# B&R Automation Studio project Nitto (part 15)

#### FB_CrossCutter.st
```iecst
//(********************************************************************
// * COPYRIGHT -- Microsoft
// ********************************************************************
// * Programm: MAIN
// * Datei: FB_CuttingAxis.st
// * Autor: Awalz
// * Erstellt: 19. Mai 2014
// ********************************************************************
// * Implementierung des Programms MAIN
// ********************************************************************)
//
// (*<$Description$> TODO: Bitte Kommentar hier einzufügen </$Description$>*)
FUNCTION_BLOCK FB_CrossCutter
	SetupPar.Acceleration	:= 1000000.0;
	SetupPar.Deceleration	:= 1000000.0;
	SetupPar.Velocity		:= SLS_MASTER_VELO;
	RegMarkPar.WindowNegative	:= 30000.0;
	RegMarkPar.WindowPositive	:= 30000.0;

	MC_BR_ReadAxisError_0.Axis				:= SlaveREF;
	MC_BR_ReadAxisError_0.Enable			:= NOT MC_BR_ReadAxisError_0.Error;
	MC_BR_ReadAxisError_0();

	MC_ReadStatus_0.Axis					:= SlaveREF;
	MC_ReadStatus_0.Enable					:= NOT MC_ReadStatus_0.Error;
	MC_ReadStatus_0();
	MC_BR_ReadDriveStatus_0.Axis			:= SlaveREF;
	MC_BR_ReadDriveStatus_0.AdrDriveStatus	:= ADR(DriveStatus);
	MC_BR_ReadDriveStatus_0.Enable			:= NOT MC_BR_ReadDriveStatus_0.Error;
	MC_BR_ReadDriveStatus_0();

	MC_ReadActualPosition_0.Axis			:= SlaveREF;
	MC_ReadActualPosition_0.Enable			:= Enable;
	MC_ReadActualPosition_0();

	MC_Reset_0.Axis	:= SlaveREF;
	MC_Reset_0();

	MC_ReadParameter_AxisPeriod.Axis			:= SlaveREF;
	MC_ReadParameter_AxisPeriod.ParameterNumber	:= 1008;	//axis modulo period
	MC_ReadParameter_AxisPeriod.Enable			:= Enable;
	MC_ReadParameter_AxisPeriod();

//********************		CrossCutter			********************
	MC_BR_CrossCutterControl_0.Master									:= machineMaster.AxisREF;
	MC_BR_CrossCutterControl_0.Slave									:= SlaveREF;
	MC_BR_CrossCutterControl_0.CutRangeMaster 							:= crosscuttpar.CutRangeMaster;
	MC_BR_CrossCutterControl_0.CutRangeSlave 							:= crosscuttpar.CutRangeSlave;
	MC_BR_CrossCutterControl_0.ProductLength 							:= crosscuttpar.ProductLength;
	MC_BR_CrossCutterControl_0.AdvancedParameters.StartMode 			:= crosscuttpar.StartMode;
	MC_BR_CrossCutterControl_0.AdvancedParameters.StartInterval			:= crosscuttpar.StartInterval;
//    MC_BR_CrossCutterControl_0.AdvancedParameters.MasterStartDistance	:= crosscuttpar.MasterStartDistance;
//	MC_BR_CrossCutterControl_0();

	IF (MC_ReadParameter_AxisPeriod.Value <> 0.0) THEN
		NeutralPosition	:= fmod( (MC_BR_CrossCutterControl_0.AdvancedParameters.CutPosition + MC_ReadParameter_AxisPeriod.Value / 2.0), MC_ReadParameter_AxisPeriod.Value);
//		IS.NeutralPosition	:= 0.0;			// Stanze ist nach Referenzfahrt in Position
	ELSE
		NeutralPosition	:= 0.0;
	END_IF;

	//**********************	START OF STATE MACHINE	**************************
	//**********************	transitions from any state	**********************
	IF (NOT Enable) THEN
		Error		:= FALSE;
		ErrorID		:= 0;
		State	:= STATE_DISABLED;
//	ELSIF (markpoints.Error) THEN
//		ErrorID		:= markpoints.ErrorID;
//		Error		:= TRUE;
//		State	:= STATE_ERROR;
	ELSIF (MC_BR_CrossCutterControl_0.Error) THEN
		ErrorID		:= MC_BR_CrossCutterControl_0.ErrorID;
		Error		:= TRUE;
		State	:= STATE_ERROR;
//	ELSIF (MC_BR_Phasing_0.Error) THEN
//		ErrorID		:= MC_BR_Phasing_0.ErrorID;
//		Error		:= TRUE;
//		State	:= STATE_ERROR;
//	ELSIF (MC_BR_ReadAutPosition_0.Error) THEN
//		ErrorID		:= MC_BR_ReadAutPosition_0.ErrorID;
//		Error		:= TRUE;
//		State	:= STATE_ERROR;
	ELSIF (MC_MoveAbsolute_0.Error) THEN
		ErrorID		:= MC_MoveAbsolute_0.ErrorID;
		Error		:= TRUE;
		State	:= STATE_ERROR;
	ELSIF (MC_ReadParameter_AxisPeriod.Error) THEN
		ErrorID		:= MC_ReadParameter_AxisPeriod.ErrorID;
		Error		:= TRUE;
		State	:= STATE_ERROR;
	END_IF;
	//****************************************************************************

	CASE State OF
		//**********************	FUB inactive	**********************
		STATE_DISABLED:
			MC_BR_ReadAutPosition_0.Execute		:= FALSE;
			MC_MoveAbsolute_0.Execute			:= FALSE;
			MC_BR_CrossCutterControl_0.Enable	:= FALSE;
			MC_BR_CrossCutterControl_0.EnableCut:= FALSE;
			EnableRestart						:= FALSE;
			SetupComplete						:= FALSE;

			IF Enable  (*OR RestartAllowed *)THEN
				State	:= STATE_INIT;
			END_IF;
	//****************************************************************

	//**********************	Internal variables are initialized	**********************
		STATE_INIT:
			GetNextCuttPos.reset := TRUE;
			State	:= STATE_IDLE;
	//************************************************************************************

	//**********************	Waiting for a movement command	**********************
		STATE_IDLE:
			GetNextCuttPos.reset := FALSE;
			IF RestartAllowed THEN
				EnableRestart						:= TRUE;
			END_IF;
			IF (EnableMove) THEN
				MC_BR_CrossCutterControl_0.Enable	:= TRUE;
				MC_BR_CrossCutterControl_0.EnableCut:= FALSE;
				State	:= STATE_CHECK_STANDBY;
			END_IF;
	//*********************************************************************************

	//**********************	Checking if automat restart is possible	**********************
		STATE_CHECK_STANDBY:
			IF (MC_BR_CrossCutterControl_0.Active) THEN
				MC_BR_CrossCutterControl_0.Enable		:= FALSE;
				MC_BR_CrossCutterControl_0.EnableCut	:= FALSE;
				IF (MC_BR_CrossCutterControl_0.StandBy AND EnableRestart) THEN
					MC_BR_ReadAutPosition_0.Execute		:= TRUE;
					State	:= STATE_READ_AUT_POS;
				ELSE
					SetupComplete					:= FALSE;
					MC_MoveAbsolute_0.Direction		:= mcPOSITIVE_DIR;
					MC_MoveAbsolute_0.Position		:= NeutralPosition;
					//IS.MC_MoveAbsolute_0.Execute		:= TRUE;	// Keine Bewegung mehr auf die NeutralPosition
					// 2013-08-22 /scoenefeldr/
				(*	MC_BR_CrossCutterControl_0.AdvancedParameters.MasterStartDistance	:= MC_BR_CrossCutterControl_0.AdvancedParameters.CutPosition - MC_ReadActualPosition_0.Position;*)
						MC_BR_CrossCutterControl_0.AdvancedParameters.MasterStartDistance	:= MC_BR_CrossCutterControl_0.AdvancedParameters.CutPosition + MC_ReadActualPosition_0.Position;
					IF (MC_BR_CrossCutterControl_0.AdvancedParameters.MasterStartDistance < 0 OR MC_BR_CrossCutterControl_0.AdvancedParameters.MasterStartDistance < data.general.periodLength) THEN
						MC_BR_CrossCutterControl_0.AdvancedParameters.MasterStartDistance	:= (*MC_BR_CrossCutterControl_0.AdvancedParameters.MasterStartDistance + *)data.general.periodLength;
					ELSIF (MC_BR_CrossCutterControl_0.AdvancedParameters.MasterStartDistance > data.general.periodLength) THEN
						MC_BR_CrossCutterControl_0.AdvancedParameters.MasterStartDistance	:=(* MC_BR_CrossCutterControl_0.AdvancedParameters.MasterStartDistance - data.general.periodLength;*) scalePerimeter.realperimeter;
					END_IF
					State							:= STATE_MOVE_TO_NEUTRAL_POS;
				END_IF;
			END_IF;
			IF (NOT EnableMove) THEN
				MC_BR_ReadAutPosition_0.Execute		:= FALSE;
				MC_BR_CrossCutterControl_0.Enable	:= FALSE;
				MC_BR_CrossCutterControl_0.EnableCut:= FALSE;
				State	:= STATE_IDLE;
			END_IF;
	//****************************************************************************************

	//**********************	Reading automat position	**********************
		STATE_READ_AUT_POS:
			IF (MC_BR_ReadAutPosition_0.Done) THEN
				MC_BR_ReadAutPosition_0.Execute	:= FALSE;
				MC_MoveAbsolute_0.Direction		:= mcPOSITIVE_DIR + mcAUTOMAT_POS;
				MC_MoveAbsolute_0.Position		:= MC_BR_ReadAutPosition_0.AutPosition;
				MC_MoveAbsolute_0.Execute		:= TRUE;
				State							:= STATE_MOVE_TO_AUT_POS;
			END_IF;

			IF (NOT EnableMove) THEN
				MC_BR_ReadAutPosition_0.Execute	:= FALSE;
				MC_MoveAbsolute_0.Execute		:= FALSE;
				State	:= STATE_IDLE;
			END_IF;
	//*****************************************************************************

	//**********************	Moving to automat position	**********************
		STATE_MOVE_TO_AUT_POS:
			IF MC_MoveAbsolute_0.Done THEN
				MC_MoveAbsolute_0.Execute			:= FALSE;
				MC_BR_CrossCutterControl_0.AdvancedParameters.StartMode	:= mcRESTART + mcCORRECT_CURRENT_CYCLE;
				MC_BR_CrossCutterControl_0.Enable	:= TRUE;
				MC_BR_CrossCutterControl_0.EnableCut:= TRUE;
				MC_BR_CrossCutterControl_0.AdvancedParameters.MasterMaxVelocity	:= SetupPar.Velocity; (*data.general.maxVelocity;*)
				State	:= STATE_START_AUTOMAT;
			ELSIF MC_MoveAbsolute_0.CommandAborted THEN
				MC_MoveAbsolute_0.Execute			:= FALSE;
				State	:= STATE_W4_RESET;
			END_IF;

			IF NOT EnableMove THEN
				MC_MoveAbsolute_0.Execute			:= FALSE;
				MC_BR_CrossCutterControl_0.Enable	:= FALSE;
				MC_BR_CrossCutterControl_0.EnableCut:= FALSE;
				State	:= STATE_IDLE;
			END_IF;
	//*****************************************************************************

	//**********************	Moving to neutral position	**********************
		STATE_MOVE_TO_NEUTRAL_POS:
			IF (TRUE) THEN
				MC_MoveAbsolute_0.Execute			:= FALSE;
				MC_BR_CrossCutterControl_0.AdvancedParameters.StartMode	:= mcIMMEDIATE + mcCORRECT_CURRENT_CYCLE;
				MC_BR_CrossCutterControl_0.Enable	:= TRUE;
				MC_BR_CrossCutterControl_0.EnableCut:= TRUE;
				MC_BR_CrossCutterControl_0.AdvancedParameters.MasterMaxVelocity	:= SetupPar.Velocity; (*data.general.maxVelocity;*)
				State	:= STATE_START_AUTOMAT;

			ELSIF (MC_MoveAbsolute_0.CommandAborted) THEN
				MC_MoveAbsolute_0.Execute	:= FALSE;
				State	:= STATE_W4_RESET;
			END_IF;

			IF NOT EnableMove THEN
				MC_MoveAbsolute_0.Execute			:= FALSE;
				MC_BR_CrossCutterControl_0.Enable	:= FALSE;
				MC_BR_CrossCutterControl_0.EnableCut:= FALSE;
				State	:= STATE_IDLE;
			END_IF;
	//*****************************************************************************

	//**********************	Starting cam automat	**********************
		STATE_START_AUTOMAT:
			IF (MC_BR_CrossCutterControl_0.Active) THEN
				EnableRestart	:= TRUE;
				State			:= STATE_RUNNING;
			ELSIF (MC_BR_CrossCutterControl_0.CommandAborted) THEN
				MC_BR_CrossCutterControl_0.Enable	:= FALSE;
				MC_BR_CrossCutterControl_0.EnableCut:= FALSE;
				State	:= STATE_W4_RESET;
			END_IF;

			IF (NOT EnableMove) THEN
				MC_BR_CrossCutterControl_0.Enable	:= FALSE;
				MC_BR_CrossCutterControl_0.EnableCut:= FALSE;
				State	:= STATE_IDLE;
			END_IF;
	//************************************************************************

	//**********************	Cam automat is running	**********************
		STATE_RUNNING:
			IF (MC_BR_CrossCutterControl_0.CommandAborted) THEN
				MC_BR_CrossCutterControl_0.Enable	:= FALSE;
				MC_BR_CrossCutterControl_0.EnableCut:= FALSE;
				State	:= STATE_W4_RESET;
			END_IF;
//			IF RestartAllowed THEN (* um die Achse wieder zu koppeln*)
//				RestartAllowed := FALSE;
//				EnableRestart						:= TRUE;
//				MC_BR_CrossCutterControl_0.Enable	:= FALSE;
//				MC_BR_CrossCutterControl_0.EnableCut:= FALSE;
//				State	:= STATE_W4_RESET;
//			END_IF
			//cam automat synchronization movement is complete
			IF ( (MC_BR_CrossCutterControl_0.IS.AutActStIdx >= 2) AND (MC_BR_CrossCutterControl_0.IS.AutActStIdx <= 6) ) THEN
				SetupComplete	:= TRUE;
			END_IF;
			//set master speed to maximum velocity after start movement is complete
			IF (MC_BR_CrossCutterControl_0.InCompensation) THEN
				MC_BR_CrossCutterControl_0.AdvancedParameters.MasterMaxVelocity	:= SetupPar.Velocity; (*data.general.maxVelocity;;*)
			END_IF;
			IF (NOT EnableMove) THEN
				MC_BR_CrossCutterControl_0.Enable	:= FALSE;
				MC_BR_CrossCutterControl_0.EnableCut	:= FALSE;
			State	:= STATE_IDLE;
			END_IF;
	//************************************************************************

	//**********************	Command aborted, wait until "EnableMove" is reset	**********************
		STATE_W4_RESET:
			IF  EnableMove THEN
				State	:= STATE_IDLE;
			END_IF;
	//************************************************************************

	//**********************	FUB Error	**********************
		STATE_ERROR:
			(*MC_BR_CrossCutterControl_0.AdvancedParameters.MasterStartDistance	:= 0;*)
			MC_BR_CrossCutterControl_0.Enable := FALSE;
			State := STATE_CHECK_STANDBY;
	//************************************************************

		ELSE

	END_CASE;
	//**********************	END OF STATE MACHINE	************************

	(*********************		Read automat position	********************)
	MC_BR_ReadAutPosition_0.Axis		:= SlaveREF;
	MC_BR_ReadAutPosition_0();
	//******************************************************************************
	//********************		Move absolute			********************
	MC_MoveAbsolute_0.Axis			:= SlaveREF;
	MC_MoveAbsolute_0.Velocity		:= 40000;
	MC_MoveAbsolute_0.Acceleration	:= 60000;
	MC_MoveAbsolute_0.Deceleration	:= 60000;
	MC_MoveAbsolute_0();
	//*********************************************************************

	//**************************************************************************//
	//limit correction value
	LCRLimit_Correction.max_value	:= REAL_TO_DINT (data.recipe.MaxCorr);  (*AutPar.MaxCorrection;*)
	LCRLimit_Correction.min_value	:= - REAL_TO_DINT (data.recipe.MaxCorr); (* AutPar.MaxCorrection;*)

	//calculate cut position within tool segment period
	IF (MC_ReadParameter_AxisPeriod.Value <> 0.0) THEN
		MC_BR_CrossCutterControl_0.CutRangeSlave		:= DINT_TO_REAL( (crosscuttpar.CutEndPos - crosscuttpar.CutStartPos) MOD REAL_TO_DINT(MC_ReadParameter_AxisPeriod.Value) );
		IF (MC_BR_CrossCutterControl_0.CutRangeSlave < 0.0) THEN
			MC_BR_CrossCutterControl_0.CutRangeSlave	:= MC_BR_CrossCutterControl_0.CutRangeSlave + MC_ReadParameter_AxisPeriod.Value;
		END_IF
		IF 	crosscuttpar.CutStartPos > crosscuttpar.CutEndPos THEN
			MC_BR_CrossCutterControl_0.AdvancedParameters.CutPosition	:= DINT_TO_REAL((crosscuttpar.CutEndPos + crosscuttpar.CutStartPos + REAL_TO_DINT(MC_ReadParameter_AxisPeriod.Value)) / 2 MOD REAL_TO_DINT(MC_ReadParameter_AxisPeriod.Value));
		ELSE
			MC_BR_CrossCutterControl_0.AdvancedParameters.CutPosition	:= DINT_TO_REAL((crosscuttpar.CutEndPos + crosscuttpar.CutStartPos) /2 MOD REAL_TO_DINT(MC_ReadParameter_AxisPeriod.Value));
		END_IF
			IF (MC_BR_CrossCutterControl_0.AdvancedParameters.CutPosition < 0.0) THEN
			MC_BR_CrossCutterControl_0.AdvancedParameters.CutPosition	:= MC_BR_CrossCutterControl_0.AdvancedParameters.CutPosition + MC_ReadParameter_AxisPeriod.Value;
			END_IF;
		//limit cut range of slave to avoid ACOPOS errors on wrong user input
		IF ((crosscuttpar.MinCutRangeSlave > 0.0) AND (crosscuttpar.MinCutRangeSlave < MC_ReadParameter_AxisPeriod.Value)) THEN
			MC_BR_CrossCutterControl_0.CutRangeSlave	:= MAX(MC_BR_CrossCutterControl_0.CutRangeSlave, crosscuttpar.MinCutRangeSlave);
		END_IF;
		IF ((crosscuttpar.MinCompRangeSlave > 0.0) AND (crosscuttpar.MinCompRangeSlave < MC_ReadParameter_AxisPeriod.Value) ) THEN
			MC_BR_CrossCutterControl_0.CutRangeSlave := MIN(MC_BR_CrossCutterControl_0.CutRangeSlave, (MC_ReadParameter_AxisPeriod.Value - crosscuttpar.MinCompRangeSlave));
		END_IF;

		//scale cut range of master
		LCRLimScal_CutRangeMaster.x1	:= 0.0;
		LCRLimScal_CutRangeMaster.y1	:= MC_BR_CrossCutterControl_0.CutRangeSlave;
		LCRLimScal_CutRangeMaster.x2	:= 100.0;
		LCRLimScal_CutRangeMaster.y2	:= (MC_BR_CrossCutterControl_0.CutRangeSlave * crosscuttpar.ProductLength) / MC_ReadParameter_AxisPeriod.Value;
		LCRLimScal_CutRangeMaster.x		:= crosscuttpar.Insetting;
		LCRLimScal_CutRangeMaster();
		MC_BR_CrossCutterControl_0.CutRangeMaster	:= LCRLimScal_CutRangeMaster.y;
	ELSE
		MC_BR_CrossCutterControl_0.CutRangeSlave					:= 0.0;
		MC_BR_CrossCutterControl_0.CutRangeMaster					:= 0.0;
		MC_BR_CrossCutterControl_0.AdvancedParameters.CutPosition	:= 0.0;
	END_IF;
	//******************************************************************
	//choose source of reg mark correction
	GetNextCuttPos( scalePerimeter := scalePerimeter, markpoints := markpoints, machinemaster := machineMaster);

	IF (RegMarkPar.EnableRmCorrection) THEN
		IF (RegMarkPar.EnableVRegMark) THEN
			LCRLimit_Correction.in	:= GetNextCuttPos.setCutOffset.setOffset_o;
			syncFtrig(CLK := MC_BR_CrossCutterControl_0.InCut);
			IF syncFtrig.Q THEN
				initdata := TRUE;
			END_IF
			(*Steckung bzw. Stauchung der Länge;*)
			IF MC_BR_CrossCutterControl_0.CutCount  <>  CutCount_1 AND initdata THEN
				CutCount_1 := MC_BR_CrossCutterControl_0.CutCount;
				MC_BR_CrossCutterControl_0.InitData	:= TRUE;
				initdata := FALSE;
			END_IF
		ELSE
			LCRLimit_Correction.in	:= GetNextCuttPos.PositionError;
//			syncFtrig(CLK := MC_BR_CrossCutterControl_0.InCut);
//			IF syncFtrig.Q THEN
//				initdata := TRUE;
//			END_IF

			syncRtrig(CLK := MC_BR_CrossCutterControl_0.InCut);
			IF MC_BR_CrossCutterControl_0.CutCount <> CutCntOld THEN
				initdata := TRUE;
				CutCntOld := MC_BR_CrossCutterControl_0.CutCount;
			END_IF
			IF  markpoints.ProbeCounter  <>  CutCount_1 AND markpoints.ProbeCounter < 1 AND initdata THEN
				CutCount_1 := markpoints.ProbeCounter;
				MC_BR_CrossCutterControl_0.InitData	:= TRUE;
				initdata := FALSE;
			ELSIF markpoints.ProbeCounter > 1 AND initdata THEN
				MC_BR_CrossCutterControl_0.InitData	:= TRUE;
				initdata := FALSE;
			END_IF
//			R_TRIG_InCompensation(CLK := MC_BR_CrossCutterControl_0.InCompensation);
//			IF R_TRIG_InCompensation.Q THEN
//				initdata := TRUE;
//			END_IF
//			IF  GetNextCuttPos.newdata <>  CutCount_1 AND  NOT MC_BR_CrossCutterControl_0.InCut(*AND initdata*) THEN
//				CutCount_1 := GetNextCuttPos.newdata;
//				MC_BR_CrossCutterControl_0.InitData	:= TRUE;
//				initdata := FALSE;
//			END_IF
		END_IF;
	ELSE
		LCRLimit_Correction.in	:= 0.0;
	END_IF;
	LCRLimit_Correction();	(*markpoints.CorrectionValid *)
	MC_BR_CrossCutterControl_0.ProductLengthCorrection	:= LCRLimit_Correction.out;
	IF MC_BR_CrossCutterControl_0.InitData THEN
		(*MC_BR_CrossCutterControl_0.ProductLengthCorrection	:= LCRLimit_Correction.out;*)
		OffsetValue1 := REAL_TO_DINT (MC_BR_CrossCutterControl_0.ProductLengthCorrection);
	END_IF
	MC_BR_CrossCutterControl_0();
	markpoints();
	IF MC_BR_CrossCutterControl_0.DataInitialized THEN
		MC_BR_CrossCutterControl_0.InitData	:= FALSE;
	END_IF
	Active				:= MC_BR_CrossCutterControl_0.Active;
	CutMasterPosition	:= MC_BR_CrossCutterControl_0.CutMasterPosition;
	RegMarkPar.Axis 	:= SlaveREF;
	//probe counter
	(*markpoints();*)
	ProbeCounter		:= markpoints.ProbeCounter;
	MissedTriggers		:= markpoints.MissedTriggers;
	ActPositionError	:= markpoints.CorrectionValue;
	IF (Enable AND RegMarkPar.EnableRmCorrection) THEN
		IF (RegMarkPar.EnableVRegMark) THEN
			ProbeCounter		:= ProbeCounter + BOOL_TO_UDINT(SPR_RmCalcPosError_Virtual.RecordedValueValid);
			MissedTriggers		:= 0;
			ActPositionError	:= PositionError;
		ELSE

		END_IF;
	ELSE
		ProbeCounter		:= 0;
		MissedTriggers		:= 0;
		ActPositionError	:= 0;
	END_IF;
END_FUNCTION_BLOCK
```

#### ac_manualCU.st
```iecst
(********************************************************************
 * COPYRIGHT -- Microsoft
 ********************************************************************
 * Programm: MAIN
 * Datei: ac_manualCU.st
 * Autor: Awalz
 * Erstellt: 21. Mai 2014
 ********************************************************************
 * Implementierung des Programms MAIN
 ********************************************************************)

 (*<$Description$> Fügt eine neue Aktion zum IEC Programm oder Bibliothek </$Description$>*)
ACTION ac_manualCU:
	status.isCoupled := axis.ctrl.MC_ReadStatus_0.SynchronizedMotion;

	CASE state OF
		ST_IDLE:

			IF status.dataOk THEN
				IF data.newTools OR data.newRecipe THEN
					IF data.recipe.mode = CONST.CUTTINGUNIT.MODEs.DISABLE THEN
						modeCtrl.mode := data.recipe.mode;
						config (cmd := CONST.CUTTINGUNIT.CMDs.DEINIT, machineMaster := machineMaster,axis := axis, status := status, data := data,
						IOs := IOs, powerbridge := powerbridge, scalePerimeter := scalePerimeter,markpoints := markpoints, camtable := camtable,  getNextUnitSyncPos := getNextUnitSyncPos, setCutOffset := setCutOffset);
						busy := TRUE;
						state := ST_SETDATA_WAIT;
					ELSE
						modeCtrl.mode := data.recipe.mode;
						check(machdata := data.machdata, recipe := data.recipe, general := data.general, modeCtrl := modeCtrl);
						IF check.err.flag THEN
							data.err := check.err;
						ELSE
							config (cmd := CONST.CUTTINGUNIT.CMDs.SETDATA, machineMaster := machineMaster, axis := axis, status := status, data := data,
							IOs := IOs, powerbridge := powerbridge, scalePerimeter := scalePerimeter,markpoints := markpoints, camtable := camtable,  getNextUnitSyncPos := getNextUnitSyncPos, setCutOffset := setCutOffset);
							state := ST_SETDATA_WAIT;
						END_IF
					END_IF
				ELSE
					IF data.recipe.mode = CONST.CUTTINGUNIT.MODEs.DISABLE THEN // Stanzen dennoch bewegen können*)

						IF cmdCtrl.value = CONST.CUTTINGUNIT.CMDs.MOVEFW OR cmdCtrl.value = CONST.CUTTINGUNIT.CMDs.MOVEBW THEN
							cmdStatus(set := TRUE, value := cmdCtrl.value);
							busy := TRUE;
							state := ST_MOVE_START;
						ELSIF cmdCtrl.value <> CONST.CUTTINGUNIT.CMDs.NO_CMD AND NOT cmdCtrl.value = CONST.CUTTINGUNIT.CMDs.RESET THEN
							cmdStatus(set := TRUE, value := cmdCtrl.value);
							busy := TRUE;
							state := ST_FUNCTION_START;
						END_IF
					ELSE
						IF NOT status.isCalibrated OR NOT axis.ctrl.BasicControl.AxisState.Homed THEN
							modeCtrl.mode := data.recipe.mode;
							IF cmdCtrl.value = CONST.CUTTINGUNIT.CMDs.CALIBR THEN (*warten bis das kommando  gesetzt wird*)
								cmdStatus(set := TRUE, value := cmdCtrl.value);
								busy := TRUE;
								state := ST_FUNCTION_START;
							ELSIF cmdCtrl.value = CONST.CUTTINGUNIT.CMDs.MOVEFW OR cmdCtrl.value = CONST.CUTTINGUNIT.CMDs.MOVEBW THEN
								cmdStatus(set := TRUE, value := cmdCtrl.value);
								busy := TRUE;
								state := ST_MOVE_START;
							END_IF
						ELSE
							IF cmdCtrl.value = CONST.CUTTINGUNIT.CMDs.MOVEFW OR cmdCtrl.value = CONST.CUTTINGUNIT.CMDs.MOVEBW THEN
								cmdStatus(set := TRUE, value := cmdCtrl.value);
								busy := TRUE;
								state := ST_MOVE_START;
							ELSIF cmdCtrl.value = CONST.CUTTINGUNIT.CMDs.CALIBR THEN
								cmdStatus(set := TRUE, value := cmdCtrl.value);
								busy := TRUE;
								state := ST_FUNCTION_QUIT;
							ELSIF cmdCtrl.value = CONST.CUTTINGUNIT.CMDs.SYNC THEN
								cmdStatus(set := TRUE, value := cmdCtrl.value);
								busy := TRUE;
								state := ST_FUNCTION_START;
							ELSIF cmdCtrl.value = CONST.CUTTINGUNIT.CMDs.CPL_ON THEN// manuell koppeln
								cmdStatus(set := TRUE, value := cmdCtrl.value);
								busy := TRUE;
								state := ST_FUNCTION_START;
							ELSIF manualFirst AND axis.ctrl.MC_ReadStatus_0.StandStill THEN//bei Steuerung Aus/Ein wieder einkoppeln
								busy := TRUE;
								manualFirst := FALSE;
								state := ST_CPLON_WAIT;
							END_IF
						END_IF
					END_IF
				END_IF
			END_IF

		ST_CPLON_WAIT:
			IF config.busy THEN
				config(cmd := CONST.CUTTINGUNIT.CMDs.NO_CMD, machineMaster := machineMaster, axis := axis, status := status,data := data,
				IOs := IOs, powerbridge := powerbridge, scalePerimeter := scalePerimeter,markpoints := markpoints, camtable := camtable,  getNextUnitSyncPos := getNextUnitSyncPos, setCutOffset := setCutOffset);
			ELSE
				config(cmd := CONST.CUTTINGUNIT.CMDs.CPL_ON, machineMaster := machineMaster, axis := axis, status := status,data := data,
				IOs := IOs, powerbridge := powerbridge, scalePerimeter := scalePerimeter,markpoints := markpoints, camtable := camtable,  getNextUnitSyncPos := getNextUnitSyncPos, setCutOffset := setCutOffset);
				state := ST_FUNCTION;
			END_IF

		ST_SETDATA_WAIT:
			config ( machineMaster := machineMaster, axis := axis, status := status, data := data, IOs := IOs, powerbridge := powerbridge,
				scalePerimeter := scalePerimeter, markpoints := markpoints, camtable := camtable,  getNextUnitSyncPos := getNextUnitSyncPos, setCutOffset := setCutOffset);
			IF NOT config.busy THEN
				IF config.err.flag THEN
					err := config.err;
					err.state := state;
					state := ST_ERROR;
				ELSE
					tmpData(set := TRUE, setMasterModulData := data.general, setMach := data.machdata, setRecipe := data.recipe, BetrCtrl := BetrCtrl );
					data(newRecipe := FALSE, newMach := FALSE);
					busy := FALSE;
					config(cmd := CONST.CUTTINGUNIT.CMDs.NO_CMD, machineMaster := machineMaster, axis := axis, status := status,data := data,
					IOs := IOs, powerbridge := powerbridge, scalePerimeter := scalePerimeter,markpoints := markpoints, camtable := camtable,  getNextUnitSyncPos := getNextUnitSyncPos, setCutOffset := setCutOffset);
					state := ST_IDLE;
				END_IF
			ELSIF  cmdCtrl.value = CONST.CUTTINGUNIT.CMDs.RESET THEN //14.04.15
				config(cmd := CONST.CUTTINGUNIT.CMDs.RESET, machineMaster := machineMaster, axis := axis, status := status, data := data,
				IOs := IOs, powerbridge := powerbridge, scalePerimeter := scalePerimeter,markpoints := markpoints, camtable := camtable,  getNextUnitSyncPos := getNextUnitSyncPos, setCutOffset := setCutOffset);
				state := ST_FUNCTION_ABORT_WAIT;
			END_IF

		ST_FUNCTION_START:
			IF config.busy OR config.cmd <> CONST.CUTTINGUNIT.CMDs.NO_CMD THEN
				config(cmd := CONST.CUTTINGUNIT.CMDs.NO_CMD, machineMaster := machineMaster, axis := axis, status := status, data := data,
				IOs := IOs, powerbridge := powerbridge, scalePerimeter := scalePerimeter, markpoints := markpoints, camtable := camtable,  getNextUnitSyncPos := getNextUnitSyncPos, setCutOffset := setCutOffset);
			ELSE
				config (cmd := cmdStatus.value, machineMaster := machineMaster, axis := axis, status := status, data := data, IOs := IOs,
				powerbridge := powerbridge, scalePerimeter := scalePerimeter, markpoints := markpoints, camtable := camtable,  getNextUnitSyncPos := getNextUnitSyncPos, setCutOffset := setCutOffset);
				state := ST_FUNCTION;
			END_IF

		ST_FUNCTION://12
			config(machineMaster := machineMaster, axis := axis, status := status, data := data, IOs := IOs, powerbridge := powerbridge,
				scalePerimeter := scalePerimeter, markpoints := markpoints, camtable := camtable, getNextUnitSyncPos := getNextUnitSyncPos, setCutOffset := setCutOffset);
			IF cmdCtrl.value = CONST.CUTTINGUNIT.CMDs.ABORT THEN
				config(cmd := CONST.CUTTINGUNIT.CMDs.ABORT, machineMaster := machineMaster, axis := axis, status := status, data := data,
				IOs := IOs, powerbridge := powerbridge, scalePerimeter := scalePerimeter, markpoints := markpoints, camtable := camtable,  getNextUnitSyncPos := getNextUnitSyncPos, setCutOffset := setCutOffset);
				state := ST_FUNCTION_ABORT_WAIT;
			ELSIF NOT config.busy THEN
				IF config.err.flag THEN
					err := config.err;
					err.state := state;
				END_IF
				config(cmd := CONST.CUTTINGUNIT.CMDs.NO_CMD, machineMaster := machineMaster, axis := axis, status := status, data := data,
				IOs := IOs, powerbridge := powerbridge, scalePerimeter := scalePerimeter,markpoints := markpoints, camtable := camtable,  getNextUnitSyncPos := getNextUnitSyncPos, setCutOffset := setCutOffset);
				state := ST_FUNCTION_QUIT;
			ELSIF (*config.err.flag AND*) cmdCtrl.value = CONST.CUTTINGUNIT.CMDs.RESET THEN //14.04.15
				config(cmd := CONST.CUTTINGUNIT.CMDs.RESET, machineMaster := machineMaster, axis := axis, status := status, data := data,
				IOs := IOs, powerbridge := powerbridge, scalePerimeter := scalePerimeter,markpoints := markpoints, camtable := camtable,  getNextUnitSyncPos := getNextUnitSyncPos, setCutOffset := setCutOffset);
				state := ST_FUNCTION_ABORT_WAIT;
			END_IF

		ST_FUNCTION_ABORT_WAIT:
			config( machineMaster := machineMaster, axis := axis, status := status, data := data,IOs := IOs, powerbridge := powerbridge,
				scalePerimeter := scalePerimeter, markpoints := markpoints, camtable := camtable,  getNextUnitSyncPos := getNextUnitSyncPos, setCutOffset := setCutOffset);
			IF NOT config.busy THEN
				IF config.err.flag THEN
					err := config.err;
					err.state := state;
				END_IF
				config(cmd := CONST.CUTTINGUNIT.CMDs.NO_CMD, machineMaster := machineMaster, axis := axis, status := status, data := data,
				IOs := IOs, powerbridge := powerbridge, scalePerimeter := scalePerimeter,markpoints := markpoints, camtable := camtable,  getNextUnitSyncPos := getNextUnitSyncPos, setCutOffset := setCutOffset);
				state := ST_FUNCTION_QUIT;
			END_IF

		ST_FUNCTION_QUIT:
			busy := FALSE;
			IF cmdCtrl.value = CONST.CUTTINGUNIT.CMDs.NO_CMD THEN
				cmdStatus(set := TRUE, value := CONST.CUTTINGUNIT.CMDs.NO_CMD);
				state := ST_IDLE;
			END_IF

		ST_MOVE_START:

			IF config.busy OR config.cmd <> CONST.CUTTINGUNIT.CMDs.NO_CMD THEN //27.04.15
				config(cmd := CONST.CUTTINGUNIT.CMDs.NO_CMD, machineMaster := machineMaster, axis := axis, status := status, data := data, IOs := IOs, powerbridge := powerbridge,
				scalePerimeter := scalePerimeter, markpoints := markpoints, camtable := camtable, getNextUnitSyncPos := getNextUnitSyncPos,setCutOffset := setCutOffset);
			ELSIF NOT config.busy THEN //27.04.15
				config(cmd := cmdStatus.value, machineMaster := machineMaster, axis := axis, status := status, data := data, IOs := IOs, powerbridge := powerbridge,
				scalePerimeter := scalePerimeter, markpoints := markpoints, camtable := camtable,getNextUnitSyncPos := getNextUnitSyncPos,setCutOffset := setCutOffset);
				state := ST_MOVE;
			END_IF

		ST_MOVE:
			config(machineMaster := machineMaster, axis := axis, status := status, data := data, IOs := IOs, powerbridge := powerbridge,
				scalePerimeter := scalePerimeter, markpoints := markpoints, camtable := camtable,  getNextUnitSyncPos := getNextUnitSyncPos, setCutOffset := setCutOffset);
			IF cmdCtrl.value = CONST.CUTTINGUNIT.CMDs.NO_CMD THEN
				config(cmd := CONST.CUTTINGUNIT.CMDs.NO_CMD, machineMaster := machineMaster, axis := axis, status := status, data := data,
				IOs := IOs, powerbridge := powerbridge, scalePerimeter := scalePerimeter, markpoints := markpoints, camtable := camtable,  getNextUnitSyncPos := getNextUnitSyncPos, setCutOffset := setCutOffset);
				state := ST_MOVE_QUIT;

			ELSE
				config(cmd := cmdStatus.value, machineMaster := machineMaster, axis := axis, status := status, data := data,
				IOs := IOs, powerbridge := powerbridge, scalePerimeter := scalePerimeter, markpoints := markpoints,camtable := camtable,  getNextUnitSyncPos := getNextUnitSyncPos, setCutOffset := setCutOffset);
			END_IF

		ST_MOVE_QUIT:
			config(cmd := CONST.CUTTINGUNIT.CMDs.NO_CMD, machineMaster := machineMaster, axis := axis, status := status, data := data,
			IOs := IOs, powerbridge := powerbridge, scalePerimeter := scalePerimeter, markpoints := markpoints, camtable := camtable,  getNextUnitSyncPos := getNextUnitSyncPos, setCutOffset := setCutOffset);
			IF NOT config.busy THEN
				busy := FALSE;
				cmdStatus(set := TRUE, value := CONST.CUTTINGUNIT.CMDs.NO_CMD);
				state := ST_IDLE;
			ELSIF cmdCtrl.value = CONST.CUTTINGUNIT.CMDs.RESET THEN //14.04.15
				config(cmd := CONST.CUTTINGUNIT.CMDs.RESET, machineMaster := machineMaster, axis := axis, status := status, data := data,
				IOs := IOs, powerbridge := powerbridge, scalePerimeter := scalePerimeter,markpoints := markpoints, camtable := camtable,  getNextUnitSyncPos := getNextUnitSyncPos, setCutOffset := setCutOffset);
				state := ST_FUNCTION_ABORT_WAIT;
			END_IF

		ST_ERROR:
			err.set := TRUE;
			busy := FALSE;
			IF cmdCtrl.value <> CONST.CUTTINGUNIT.CMDs.NO_CMD THEN
				err(reset := TRUE);
				state := ST_IDLE;
			ELSIF BetrCtrl.value <> CONST.MACHINEMODES.MANUAL THEN
				state := ST_IDLE;
				err(reset := TRUE);
				busy := TRUE;
				StateCtrl := CTRL_MANUAL_AFTER;
			END_IF
	END_CASE

END_ACTION
```

#### ac_cyclicCuttingCtrl.st
```iecst
(********************************************************************
 * COPYRIGHT -- Microsoft
 ********************************************************************
 * Programm: MAIN
 * Datei: ac_cyclicCuttingCtrl.st
 * Autor: awalz
 * Erstellt: 25. Juli 2014
 ********************************************************************
 * Implementierung des Programms MAIN
 ********************************************************************)

(* Fügt eine neue Aktion zum IEC Programm oder Bibliothek *)
ACTION ac_cyclicCuttingCtrl:
	markpoints.TriggerInput.Edge			:= ncP_EDGE;
	markpoints.TriggerInput.EventSourceParID:= ACP10PAR_STAT_TRIGGER1;
	markpoints.TriggerInput.MaxWidth		:= 0;
	markpoints.TriggerInput.MinWidth		:= 0;
	markpoints.TriggerInput.ProbeParID		:= ACP10PAR_MA1_CYCLIC_POS;
	markpoints.TriggerInput.SensorDelay	:= -900;
//	getNextCuttPos.setCutOffset.maxcorrection :=  REAL_TO_UDINT(data.general.periodLength /2);
//	getNextCuttPos.ProductLength := REAL_TO_UDINT(data.general.periodLength);
//	getNextCuttPos.DistanceToSensor := data.machdata.position; (*540000;*)
//	axis.ctrl();
//	cmdCtrl();
//	emcy_inputs();
//	status.isCoupled := axis.ctrl.MC_ReadStatus_0.SynchronizedMotion;
//	status(dataOk := data.loaded, recipeMode := data.recipe.mode, axisState := axis.ctrl.MC_ReadStatus_0);
//	scalePerimeter.realperimeter := UINT_TO_REAL (data.recipe.tool.cogCutting )* data.recipe.tool.cogmodul;
//	scalePerimeter.NumberToolSegments := MAX (1, data.recipe.tool.numberToolSegments);
//	scalePerimeter();
//
//	IF ABS (getNextCuttPos.PositionError) < 5000 THEN
//		status.isSynchronized := TRUE;
//	ELSE
//		status.isSynchronized := FALSE;
//	END_IF
//	IF powerbridge.movebutton.LDT.button THEN
//		cmdCtrl.value := CONST.CUTTINGUNIT.CMDs.MOVEFW;
//	ELSIF  powerbridge.movebutton.LDT.ftrig.Q THEN
//		cmdCtrl.value := CONST.CUTTINGUNIT.CMDs.NO_CMD;
//	END_IF
//	status.errorstop := axis.ctrl.MC_ReadStatus_0.Errorstop;
//	IF cmdCtrl.value = CONST.CUTTINGUNIT.CMDs.RESET AND axis.ctrl.MC_ReadStatus_0.Errorstop THEN
//		axis.ctrl.cmd := CONST.AXIS.RESET;
//	ELSIF cmdCtrl.value = CONST.CUTTINGUNIT.CMDs.RESET AND axis.ctrl.MC_ReadStatus_0.Disabled THEN
//		axis.ctrl.cmd := CONST.AXIS.POWER_ON;
//	END_IF
////////////////////////////////////////////TRIGGER füür den Touchprobe/////////////////////
//	Trigger.Axis						:= axis.ctrl.AxisREF; (*machineMaster.AxisREF;*)
//	Trigger.PositionSensor				:= data.machdata.position;
//	Trigger.TriggerInput.Edge			:= ncP_EDGE;
//	Trigger.TriggerInput.EventSourceParID:= ACP10PAR_STAT_TRIGGER1;
//	Trigger.TriggerInput.MaxWidth		:= 0; (*data.recipe.RmWindow;*)
//	Trigger.TriggerInput.MinWidth		:= 0;(*-data.recipe.RmWindow;*)
//	Trigger.TriggerInput.ProbeParID		:= ACP10PAR_MA1_CYCLIC_POS;
//	Trigger.TriggerInput.SensorDelay	:= -900;
//	markpoints.Axis    					:= axis.ctrl.AxisREF; (*machineMaster.AxisREF;*)
////	markpoints.DistanceToSensor			:= data.machdata.position; (* Distanz zum zwischen Schneidposition und dem Sensor*)
//	markpoints.ProductLength			:= data.general.periodLength;
//	markpoints.TriggerInput				:= Trigger.TriggerInput;(*wird in der Main bereits zugewiesen*)
//	markpoints.WindowNegative			:= data.recipe.RmWindow;(*- data.recipe.RmWindow;*)
//	markpoints.WindowPositive			:= data.recipe.RmWindow;
//	(*markpoints.RegMarkPosition  := usercorrection; (* Offset des Schnitts von der VISU*)
//	markpoints.Enable			:= TRUE;
//	markpoints();
//
//
////	data.check(general := data.general, machdata := data.machdata, modeCtrl := modeCtrl, recipe := data.recipe);
//	powerbridge (clk := clk);

	scalePerimeter.realperimeter := UINT_TO_REAL (data.recipe.tool.cogCutting )* data.recipe.tool.cogmodul;
	scalePerimeter.NumberToolSegments := MAX (1, data.recipe.tool.numberToolSegments);
	scalePerimeter();
	setCutOffset( enable := TRUE, maxcorrection := data.recipe.MaxCorr, limitvisupos := data.general.periodLength/1000, limitvisuneg := -data.general.periodLength/1000);
	axis.ctrl();
	cmdCtrl();
	emcy_inputs();
	//	status.isCoupled := axis.ctrl.MC_ReadStatus_0.SynchronizedMotion;
	status(dataOk := data.loaded, recipeMode := data.recipe.mode,
	axisState := axis.ctrl.MC_ReadStatus_0);
	scalePerimeter(realperimeter := UINT_TO_REAL (data.recipe.tool.cogCutting) * data.recipe.tool.cogmodul,
	NumberToolSegments := MAX (1,data.recipe.tool.numberToolSegments));
	IF emcy_inputs.EMCY_Door1 AND emcy_inputs.EMCY_Door2 THEN
		emcy_inputs.EMCY_DoorsClosed := TRUE;
	ELSE
		emcy_inputs.EMCY_DoorsClosed := FALSE;
	END_IF

	IF  status.isCalibrated AND NOT config.busy AND axis.ctrl.MC_ReadStatus_0.SynchronizedMotion THEN
		modeCtrl(machineMaster := machineMaster, mode := data.recipe.mode, axis := axis, getNextUnitSyncPos := getNextUnitSyncPos, data:= data, status := status, scalePerimeter := scalePerimeter,
		markpoints := markpoints, syncData := getNextUnitSyncPos.syncDataBefore, camCtrl := camCtrl , setCutOffset := setCutOffset);
	ELSIF cmdCtrl.value = CONST.CUTTINGUNIT.CMDs.RESET THEN
		modeCtrl(machineMaster := machineMaster, mode := CONST.CUTTINGUNIT.MODEs.DISABLE, axis := axis, getNextUnitSyncPos := getNextUnitSyncPos, data:= data, status := status, scalePerimeter := scalePerimeter,
		markpoints := markpoints, syncData := getNextUnitSyncPos.syncDataBefore, camCtrl := camCtrl , setCutOffset := setCutOffset);
	ELSE
		modeCtrl(machineMaster := machineMaster, mode := CONST.CUTTINGUNIT.MODEs.DISABLE, axis := axis, getNextUnitSyncPos := getNextUnitSyncPos, data:= data, status := status, scalePerimeter := scalePerimeter,
		markpoints := markpoints, syncData := getNextUnitSyncPos.syncDataBefore, camCtrl := camCtrl , setCutOffset := setCutOffset);
	END_IF
//
//	IF ABS (getNextCuttPos.PositionError) < 5000 THEN
//		status.isSynchronized := TRUE;
//	ELSE
//		status.isSynchronized := FALSE;
//	END_IF

	IF powerbridge.movebutton.LDT.button THEN
		cmdCtrl.value := CONST.CUTTINGUNIT.CMDs.MOVEFW;
	ELSIF  powerbridge.movebutton.LDT.ftrig.Q THEN
		cmdCtrl.value := CONST.CUTTINGUNIT.CMDs.NO_CMD;
	END_IF
	status.errorstop := axis.ctrl.MC_ReadStatus_0.Errorstop;
	IF (cmdCtrl.value = CONST.CUTTINGUNIT.CMDs.RESET OR panel.LDTRESET.LDT.button) AND axis.ctrl.MC_ReadStatus_0.Errorstop THEN
		axis.ctrl.Cmd := CONST.AXIS.RESET;
	ELSIF (cmdCtrl.value = CONST.CUTTINGUNIT.CMDs.RESET OR panel.LDTRESET.LDT.button)AND axis.ctrl.MC_ReadStatus_0.Disabled THEN
		axis.ctrl.Cmd := CONST.AXIS.POWER_ON;
	END_IF

	//	(*markpoints.RegMarkPosition  := usercorrection; (* Offset des Schnitts von der VISU*)
	markpoints(Axis	:= axis.ctrl.AxisREF, Enable:= TRUE,
	ProductLength 	:= data.general.periodLength,
	WindowNegative 	:= data.recipe.RmWindow,
	WindowPositive	:= data.recipe.RmWindow);
	powerbridge ((*enable := TRUE,*) clk := clk);
END_ACTION
```

#### FB_CuttingCtrl.st
```iecst
(********************************************************************
 * COPYRIGHT -- Microsoft
 ********************************************************************
 * Programm: MAIN
 * Datei: FB_CuttingCtrl.st
 * Autor: Awalz
 * Erstellt: 19. Mai 2014
 ********************************************************************
 * Implementierung des Programms MAIN
 ********************************************************************)

 (*<$Description$> TODO: Bitte Kommentar hier einzufügen </$Description$>*)
FUNCTION_BLOCK FB_CuttingCtrl
	ac_cyclicCuttingCtrl;
//	getNextUnitSyncPos( uData := data, machineMaster := machineMaster, markpoints := markpoints,
//						uAxis := axis.ctrl, scalePerimeter := scalePerimeter, setCutOffset :=setCutOffset, CONST :=CONST);
	CASE StateCtrl OF
	CTRL_FIRST_START:
		busy := TRUE;
		StateCtrl := CTRL_EMERGENCYSTOP_BEFORE;

	CTRL_MANUAL_BEFORE:
		IF BetrCtrl.value = CONST.MACHINEMODES.MANUAL THEN
		(*	clamp.init(clk := clk);*)
			BetrStatus(set := TRUE, value := CONST.MACHINEMODES.MANUAL);
			modeCtrl.mode  := data.recipe.mode;
			chkStatus.enable := TRUE;
			err(reset := TRUE);
			busy := FALSE;
			timer(IN:= FALSE);
			state := ST_IDLE;
			manualFirst := TRUE;
			StateCtrl := CTRL_MANUAL;
		ELSIF BetrCtrl.value = CONST.MACHINEMODES.EMERGENCYSTOP THEN
			StateCtrl := CTRL_EMERGENCYSTOP_BEFORE;
		ELSIF BetrCtrl.value = CONST.MACHINEMODES.SAFETYSTOP THEN
			StateCtrl := CTRL_SAFETYSTOP_BEFORE;
		ELSIF BetrCtrl.value = CONST.MACHINEMODES.AUTOMATIC THEN
			StateCtrl := CTRL_AUTO_BEFORE;
		END_IF

	CTRL_MANUAL://11
		IF BetrCtrl.value <> CONST.MACHINEMODES.MANUAL THEN
			err(reset := TRUE);
			busy := TRUE;
			state := ST_IDLE;
			config(cmd := CONST.CUTTINGUNIT.CMDs.NO_CMD, machineMaster := machineMaster, axis := axis, status := status,data := data,
					IOs := IOs, powerbridge := powerbridge, scalePerimeter := scalePerimeter,markpoints := markpoints, camtable := camtable,
					getNextUnitSyncPos := getNextUnitSyncPos, setCutOffset := setCutOffset);
			StateCtrl := CTRL_MANUAL_AFTER;
		ELSE
			ac_manualCU;
		END_IF

	CTRL_MANUAL_AFTER://12
			timer(IN:= FALSE);
//			state := ST_IDLE;
			chkStatus.enable := FALSE;

/////////////////////////geaendert um die Stanze automatiech zu koppeln
//			config (cmd := CONST.CUTTINGUNIT.CMDs.CPL_ON, machineMaster := machineMaster,axis := axis, status := status, data := data,
//			IOs := IOs, powerbridge := powerbridge, scalePerimeter := scalePerimeter, getNextCuttPos := getNextCuttPos);
		(*	IF NOT config.busy AND NOT  config.copple THEN*)
				ac_setStateAfterPB;
//			END_IF

	CTRL_AUTO_BEFORE:
		IF BetrCtrl.value = CONST.MACHINEMODES.AUTOMATIC THEN
		BetrStatus(set := TRUE, value := CONST.MACHINEMODES.AUTOMATIC);
			(*clamp.init(clk := clk);*)
			err(reset := TRUE);
			modeCtrl.mode  := data.recipe.mode;
			chkStatus.enable := TRUE;
			busy := FALSE;
			state := ST_IDLE;
			StateCtrl := CTRL_AUTO;
		ELSIF BetrCtrl.value = CONST.MACHINEMODES.EMERGENCYSTOP THEN
			StateCtrl := CTRL_EMERGENCYSTOP_BEFORE;
		ELSIF BetrCtrl.value = CONST.MACHINEMODES.SAFETYSTOP THEN
			StateCtrl := CTRL_SAFETYSTOP_BEFORE;
		ELSIF BetrCtrl.value = CONST.MACHINEMODES.MANUAL THEN
			StateCtrl := CTRL_MANUAL_BEFORE;
		END_IF

	(* ******************************** *)
	(* *********** AUTO *************** *)
	(* ******************************** *)
	CTRL_AUTO:
		IF BetrCtrl.value <> CONST.MACHINEMODES.AUTOMATIC THEN
			err(reset := TRUE);
			busy := TRUE;
			StateCtrl := CTRL_AUTO_AFTER;
		ELSE
		(*	modeCtrl(machineMaster := machineMaster, axis := axis, data:= data, status := status);*)
		END_IF

	CTRL_AUTO_AFTER:
		chkStatus.enable := FALSE;
		state := ST_IDLE;
		ac_setStateAfterPB;

	CTRL_STOP_BEFORE:
		IF BetrCtrl.value = CONST.MACHINEMODES.EMERGENCYSTOP THEN
			StateCtrl := CTRL_EMERGENCYSTOP_BEFORE;
		ELSIF BetrCtrl.value = CONST.MACHINEMODES.SAFETYSTOP THEN
			StateCtrl := CTRL_SAFETYSTOP_BEFORE;
		ELSE
			state := ST_IDLE;
			StateCtrl := CTRL_STOP;
		END_IF

	CTRL_STOP:
		IF BetrCtrl.value = CONST.MACHINEMODES.EMERGENCYSTOP THEN
			StateCtrl := CTRL_EMERGENCYSTOP_BEFORE;
		ELSIF BetrCtrl.value = CONST.MACHINEMODES.SAFETYSTOP THEN
			StateCtrl := CTRL_SAFETYSTOP_BEFORE;
		ELSE
			CASE state OF
			ST_IDLE:
				state := ST_QUIT;

			ST_QUIT:
				state := ST_IDLE;
				StateCtrl := CTRL_STOP_AFTER;
			END_CASE
		END_IF

	CTRL_STOP_AFTER:
		IF BetrCtrl.value = CONST.MACHINEMODES.EMERGENCYSTOP THEN
			StateCtrl := CTRL_EMERGENCYSTOP_BEFORE;
		ELSIF BetrCtrl.value = CONST.MACHINEMODES.SAFETYSTOP THEN
			StateCtrl := CTRL_SAFETYSTOP_BEFORE;
		ELSIF BetrCtrl.value = CONST.MACHINEMODES.MANUAL THEN
			StateCtrl := CTRL_MANUAL_BEFORE;
		ELSIF BetrCtrl.value = CONST.MACHINEMODES.AUTOMATIC THEN
			StateCtrl := CTRL_AUTO_BEFORE;
		END_IF

	CTRL_RESET_START:
		axis.ctrl();
		BetrStatus(set := TRUE,value := CONST.MACHINEMODES.RESET);
		modeCtrl.mode  := CONST.CUTTINGUNIT.MODEs.DISABLE;
		IF BetrCtrl.value = CONST.MACHINEMODES.EMERGENCYSTOP THEN
			StateCtrl := CTRL_EMERGENCYSTOP_BEFORE;
		ELSIF BetrCtrl.value = CONST.MACHINEMODES.SAFETYSTOP THEN
			StateCtrl := CTRL_SAFETYSTOP_BEFORE;
		ELSE
			IF axis.ctrl.busy OR axis.ctrl.Cmd <> CONST.AXIS.NOACTION THEN
				axis.ctrl.Cmd := CONST.AXIS.NOACTION;
			ELSE
				axis.ctrl.Cmd := CONST.AXIS.RESET;
				StateCtrl := CTRL_RESET;
			END_IF
		END_IF

	CTRL_RESET:
		axis.ctrl();
		(*axis.ctrl(cmd := CONST.AXIS.RESET);**********************)
		IF BetrCtrl.value = CONST.MACHINEMODES.EMERGENCYSTOP THEN
			StateCtrl := CTRL_EMERGENCYSTOP_BEFORE;
		ELSIF BetrCtrl.value = CONST.MACHINEMODES.SAFETYSTOP THEN
			StateCtrl := CTRL_SAFETYSTOP_BEFORE;
		ELSE
			(*IF NOT axis.ctrl.busy THEN*)
				modeCtrl.mode  := CONST.CUTTINGUNIT.MODEs.DISABLE;
				axis.ctrl.Cmd := CONST.AXIS.POWER_OFF;
			(*	axis.ctrl(cmd := CONST.AXIS.POWER_ON);(******************************)
				StateCtrl := CTRL_RESET_AFTER;
			(*END_IF*)
		END_IF

	CTRL_RESET_AFTER://77
		axis.ctrl();
		IF BetrCtrl.value = CONST.MACHINEMODES.RESET THEN
			busy := FALSE;
		ELSE
			busy := TRUE;
		(*	clamp.init(clk := clk);*)
			err(reset := TRUE);
			IF BetrCtrl.value = CONST.MACHINEMODES.EMERGENCYSTOP THEN
				StateCtrl := CTRL_EMERGENCYSTOP_BEFORE;
			ELSIF BetrCtrl.value = CONST.MACHINEMODES.SAFETYSTOP THEN
				StateCtrl := CTRL_SAFETYSTOP_BEFORE;
			ELSIF BetrCtrl.value = CONST.MACHINEMODES.SAFETYSTOP THEN
				StateCtrl := CTRL_SAFETYSTOP_BEFORE;
			ELSIF BetrCtrl.value = CONST.MACHINEMODES.MANUAL THEN
			(*	modeCtrl.mode  := data.recipe.mode;*)
				supplydelay(IN:= TRUE, PT := T#8s);
				IF supplydelay.Q THEN
					axis.ctrl.Cmd := CONST.AXIS.POWER_ON;
					busy := TRUE;
					supplydelay(IN:= FALSE);
					StateCtrl := CTRL_MANUAL_BEFORE;
				END_IF
			ELSIF BetrCtrl.value = CONST.MACHINEMODES.AUTOMATIC THEN
				(*modeCtrl.mode  := data.recipe.mode;*)
				supplydelay(IN:= TRUE, PT := T#8s);
				IF supplydelay.Q THEN
					axis.ctrl.Cmd := CONST.AXIS.POWER_ON;
					busy := TRUE;
					supplydelay(IN:= FALSE);
					StateCtrl := CTRL_AUTO_BEFORE;
				END_IF
			END_IF
		END_IF

	CTRL_SAFETYSTOP_BEFORE://82
			modeCtrl.mode  := CONST.CUTTINGUNIT.MODEs.DISABLE;
		IF BetrCtrl.value = CONST.MACHINEMODES.EMERGENCYSTOP THEN
			StateCtrl := CTRL_EMERGENCYSTOP_BEFORE;
		ELSE
			BetrStatus(set := TRUE,value := CONST.MACHINEMODES.SAFETYSTOP);
			state := ST_IDLE;
			axis.ctrl.Deceleration:= CONST.AXIS.EMERGENCY_DECELERATION;//11.03.15 1111111; (*200m/min in 3 sek*)
			axis.ctrl.Cmd := CONST.AXIS.STOP;
			StateCtrl := CTRL_SAFETYSTOP;
		END_IF

	CTRL_SAFETYSTOP://85
		status.isCalibrated := FALSE; // 14.01.16 OKrebs
		IF BetrCtrl.value = CONST.MACHINEMODES.EMERGENCYSTOP THEN
			StateCtrl := CTRL_EMERGENCYSTOP_BEFORE;
		ELSE
			//12.03.15
			BetrStatus(set := TRUE,value := CONST.MACHINEMODES.SAFETYSTOP);
			IF axis.ctrl.MC_ReadStatus_0.StandStill THEN
				axis.ctrl.Cmd := CONST.AXIS.POWER_OFF;
			ELSIF axis.ctrl.MC_ReadStatus_0.Disabled OR
					axis.ctrl.MC_ReadStatus_0.Errorstop OR  axis.ctrl.MC_ReadStatus_0.Error  THEN
				axis.ctrl.Cmd := CONST.AXIS.NOACTION;
				StateCtrl := CTRL_SAFETYSTOP_AFTER;
			END_IF
		END_IF

	CTRL_SAFETYSTOP_AFTER:
		busy := FALSE;
		manualFirst := TRUE;
		IF BetrCtrl.value = CONST.MACHINEMODES.EMERGENCYSTOP THEN
			busy := TRUE;
			StateCtrl := CTRL_EMERGENCYSTOP_BEFORE;
			(*modeCtrl.mode  := data.recipe.mode;*)
		ELSIF BetrCtrl.value = CONST.MACHINEMODES.MANUAL THEN
			modeCtrl.mode  := data.recipe.mode;
			supplydelay(IN:= TRUE, PT := T#8s);
			IF supplydelay.Q THEN
				axis.ctrl.Cmd := CONST.AXIS.POWER_ON;
				busy := TRUE;
				supplydelay(IN:= FALSE);
				StateCtrl := CTRL_MANUAL_BEFORE;
			END_IF

		ELSIF BetrCtrl.value = CONST.MACHINEMODES.AUTOMATIC THEN
		(*	modeCtrl.mode  := data.recipe.mode;*)
			supplydelay(IN:= TRUE, PT := T#8s);
			IF supplydelay.Q THEN
				axis.ctrl.Cmd := CONST.AXIS.POWER_ON;
				busy := TRUE;
				supplydelay(IN:= FALSE);
				StateCtrl := CTRL_AUTO_BEFORE;
			END_IF
		END_IF

	CTRL_EMERGENCYSTOP_BEFORE:
			modeCtrl.mode  := CONST.CUTTINGUNIT.MODEs.DISABLE;
		status.isCoupled := FALSE;
		IF axis.ctrl.MC_ReadStatus_0.ContinuousMotion OR axis.ctrl.MC_ReadStatus_0.DiscreteMotion
			OR axis.ctrl.MC_ReadStatus_0.SynchronizedMotion OR axis.ctrl.MC_ReadStatus_0.Homing THEN
			axis.ctrl.Deceleration := CONST.AXIS.EMERGENCY_DECELERATION; (*1666666;*) (*200m/min in 2 sek*)
			axis.ctrl.Cmd := CONST.AXIS.STOP;
			BetrStatus(set := TRUE, value := CONST.MACHINEMODES.EMERGENCYSTOP);
			StateCtrl := CTRL_EMERGENCYSTOP;
		ELSE
			axis.ctrl.Cmd := CONST.AXIS.NOACTION;
			BetrStatus(set := TRUE, value := CONST.MACHINEMODES.EMERGENCYSTOP);
			StateCtrl := CTRL_EMERGENCYSTOP;
		END_IF

	CTRL_EMERGENCYSTOP://92
		status.isCalibrated := FALSE; // 14.01.16 OKrebs
		IF BetrCtrl.value = CONST.MACHINEMODES.EMERGENCYSTOP THEN
			IF axis.ctrl.MC_ReadStatus_0.StandStill THEN
				axis.ctrl.Cmd := CONST.AXIS.POWER_OFF;
			ELSIF axis.ctrl.MC_ReadStatus_0.Disabled OR
					axis.ctrl.MC_ReadStatus_0.Errorstop OR  axis.ctrl.MC_ReadStatus_0.Error THEN
				axis.ctrl.Cmd := CONST.AXIS.NOACTION;
			END_IF
		ELSE
			busy := TRUE;
			timer(IN := TRUE, PT := T#2s);
			StateCtrl := CTRL_EMERGENCYSTOP_AFTER;
		END_IF

	CTRL_EMERGENCYSTOP_AFTER://93
		timer();
		IF BetrCtrl.value = CONST.MACHINEMODES.EMERGENCYSTOP THEN
			timer(IN := FALSE);
			BetrStatus(set := TRUE , value := CONST.MACHINEMODES.EMERGENCYSTOP);
			busy := FALSE;
			StateCtrl := CTRL_EMERGENCYSTOP;
		ELSIF timer.Q THEN
			timer(IN := FALSE);
			StateCtrl := CTRL_RESET_START;
		END_IF

	ELSE
		;
	END_CASE
//	axis.ctrl.BasicControl.Parameter.Deceleration	:= 90000.0; //only for initialization
//	axis.ctrl.BasicControl.Parameter.Acceleration	:= 90000.0;

END_FUNCTION_BLOCK
```

#### FB_CuttingConfig.st
```iecst
(********************************************************************
 * COPYRIGHT -- Microsoft
 ********************************************************************
 * Programm: MAIN
 * Datei: FB_CuttingCofig.st
 * Autor: Awalz
 * Erstellt: 19. Mai 2014
 ********************************************************************
 * Implementierung des Programms MAIN
 ********************************************************************)

 (*<$Description$> TODO: Bitte Kommentar hier einzufügen </$Description$>*)
FUNCTION_BLOCK FB_CuttingConfig
	writeEncoder( AxisREF := axis.ctrl.AxisREF, data := data, scalePerimeter := scalePerimeter);
	pAxis ACCESS axis.ctrl.AxisREF;
	axis.ctrl.BasicControl.Parameter.Deceleration	:= 120000.0;
	axis.ctrl.BasicControl.Parameter.Acceleration	:= 120000.0;

	CASE state OF
		ST_IDLE:
			IF cmd <> CONST.CUTTINGUNIT.CMDs.NO_CMD THEN
				busy := TRUE;
				err(reset := TRUE);
				cmdtmp := cmd;
				IF cmd = CONST.CUTTINGUNIT.CMDs.ABORT THEN
					state := ST_ABORT;
				ELSE
					IF cmd = CONST.CUTTINGUNIT.CMDs.CALIBR THEN   (*Referenziert die CutterAxis*)
						state := ST_INIT_START;//  ST_CALIBR_START;//  ST_SETDATA_START;//Achse referenzieren
					ELSIF cmd = CONST.CUTTINGUNIT.CMDs.INIT THEN
						state := ST_INIT_START;//Referenzsensor initialisieren, nicht beim Referenzmode mcHOME_DIRECT
					ELSIF cmd = CONST.CUTTINGUNIT.CMDs.CPL_ON THEN
						state := ST_GENERATE_TABLE_START;//Kurvenscheibe ertellen und Achse koppeln
					ELSIF cmd = CONST.CUTTINGUNIT.CMDs.SETDATA THEN
						state := ST_SETDATA_START;//Encoder initialisieren (Auflösung für die Vorschubkonstante)
					ELSIF cmd = CONST.CUTTINGUNIT.CMDs.CPL_OFF THEN
						state := ST_CPLOFF_START;//Achse stoppen damit die Achse abgekoppelt wird
					ELSIF cmd = CONST.CUTTINGUNIT.CMDs.DEINIT THEN
						state := ST_DEINIT;//Achse ausschalten
					ELSIF cmd = CONST.CUTTINGUNIT.CMDs.SYNC THEN
						state := ST_SYNC_START;//Achse synchroniesieren
					ELSIF cmd = CONST.CUTTINGUNIT.CMDs.MOVEFW OR cmd = CONST.CUTTINGUNIT.CMDs.MOVEBW THEN
						state := ST_MOVE_START;
					END_IF
				END_IF
			END_IF
		//
		ST_SETDATA_START://2
			IF axis.ctrl.MC_ReadStatus_0.StandStill  THEN
				IF NOT axis.ctrl.busy THEN
					writeEncoder.check := TRUE;
					state:= ST_SETDATA_WAIT;
				END_IF
			ELSIF status.isCoupled(*axis.ctrl.MC_ReadStatus_0.SynchronizedMotion*) THEN
				state:= ST_CPLOFF_START;
			ELSIF status.isInitialized THEN
				axis.ctrl.Cmd := CONST.AXIS.NOACTION;
				state := ST_INIT_START; //  ST_DEINIT_CPLSLAVEOFF_START;
			ELSIF axis.ctrl.MC_ReadStatus_0.Disabled THEN
				writeEncoder.InverseDirection := data.recipe.tool.addSupportSpindle;
				writeEncoder.check := TRUE;
				state:= ST_SETDATA_WAIT;
			ELSIF axis.ctrl.MC_ReadStatus_0.Errorstop THEN
				err(set := TRUE ,fnc := 'FB_CuttinConfig' ,text := 'axis.ctrl', state := ST_SETDATA_START, id := axis.ctrl.MC_BR_ReadDriveStatus_0.ErrorID);
				state := ST_ERROR;
			END_IF

		ST_SETDATA_WAIT://4
			IF (axis.ctrl.MC_ReadStatus_0.Disabled OR axis.ctrl.MC_ReadStatus_0.StandStill) AND NOT axis.ctrl.busy THEN
				writeEncoder(enable := TRUE, AxisREF := axis.ctrl.AxisREF, data := data, scalePerimeter := scalePerimeter);
				axis.ctrl.Cmd := CONST.AXIS.NOACTION;
				IF NOT writeEncoder.busy AND  NOT writeEncoder.check THEN (* Encoder initialisierung ist abgeschloßen jetzt kann referenzeirt werden*)
					status.isInitialized := TRUE;// Encoder hat neue Auflösung
					status.isSynchronized := FALSE;
					status.isCalibrated := FALSE; //nicht referenziert
					axis.ctrl.BasicControl.AxisState.Homed := FALSE;
					writeEncoder(enable := FALSE, AxisREF := axis.ctrl.AxisREF, data := data, scalePerimeter := scalePerimeter);
					IF cmd =  CONST.CUTTINGUNIT.CMDs.CALIBR AND
						(data.recipe.mode = CONST.CUTTINGUNIT.MODEs.SYNC_RUN  OR data.recipe.mode = CONST.CUTTINGUNIT.MODEs.CROSS_CUT) THEN (* wenn calibrieren dann in Init*)
						axis.ctrl.Cmd := CONST.AXIS.POWER_OFF;
						state := ST_INIT_START;
					ELSIF cmd =  CONST.CUTTINGUNIT.CMDs.CALIBR AND data.recipe.mode = CONST.CUTTINGUNIT.MODEs.FREE_RUN THEN//14.04.15
						axis.ctrl.Cmd := CONST.AXIS.POWER_ON;//15.04.15
						state := ST_CALIBR_START;
					ELSIF cmd = CONST.CUTTINGUNIT.CMDs.SETDATA THEN(* nur die Auflösung geändert*)
						cmd := CONST.CUTTINGUNIT.CMDs.NO_CMD;//15.04.15
						state := ST_QUIT;
					END_IF
				END_IF
			END_IF

		ST_INIT_START://10

			IF NOT  axis.ctrl.MC_ReadStatus_0.Disabled THEN //23.04.15
				axis.ctrl.Cmd := CONST.AXIS.POWER_OFF;
			ELSIF axis.ctrl.MC_ReadStatus_0.Disabled AND NOT axis.ctrl.busy  THEN
				axis.ctrl.Cmd := CONST.AXIS.NOACTION;
				pAxis.dig_in.level.reference := ncACTIV_HI + ncFORCE;(*initialisierung des Referenzeingamgs in der Maschine ist der Sonsor akiv low*)
				//				InitAxisSubjectPar.Axis := axis.ctrl.AxisREF; (* d.h. wenn keine Lücke dann leuchtet die SensorLed nicht*)
				InitAxisSubjectPar.Subject := ncDIG_IN;//102
				InitAxisSubjectPar.Execute := TRUE;
				IF InitAxisSubjectPar.Done THEN
					axis.refSwitchConfig(Enable := TRUE);
					InitAxisSubjectPar.Execute := FALSE;
					axis.ctrl.Cmd := CONST.AXIS.POWER_ON; //23.04.15
					state := ST_CALIBR_START;
				ELSIF InitAxisSubjectPar.Error THEN
					err.text := 'Parameter ncDIG_IN nicht initialisiert';
					err.state := state;
					state := ST_ERROR;
				END_IF
				(*END_IF*)
			END_IF

		ST_CALIBR_START: //20 (* Achse wieder einschalten*)
			//		InitAxisSubjectPar();
			axis.refSwitchConfig();
			IF axis.ctrl.MC_ReadStatus_0.Disabled THEN
				axis.ctrl.Cmd := CONST.AXIS.POWER_ON;
			ELSIF NOT axis.ctrl.busy AND axis.ctrl.MC_ReadStatus_0.StandStill AND NOT powerbridge.pressurepresent AND (data.recipe.mode = CONST.CUTTINGUNIT.MODEs.SYNC_RUN  OR data.recipe.mode = CONST.CUTTINGUNIT.MODEs.CROSS_CUT)THEN
				axis.ctrl.BasicControl.AxisState.Homed := FALSE; // falls die Achse bereits referenziert ist
				axis.ctrl.BasicControl.Parameter.HomeMode := mcHOME_SWITCH_GATE;
				axis.ctrl.BasicControl.Parameter.HomePosition := 0;
				axis.ctrl.Cmd := CONST.AXIS.CALIBR;(* Achse referenzieren*)
				state := ST_CALIBR_WAIT;
			ELSIF NOT axis.ctrl.busy AND axis.ctrl.MC_ReadStatus_0.StandStill AND NOT powerbridge.pressurepresent AND data.recipe.mode = CONST.CUTTINGUNIT.MODEs.FREE_RUN THEN
				axis.ctrl.BasicControl.AxisState.Homed := FALSE; // falls die Achse bereits referenziert ist
				axis.ctrl.BasicControl.Parameter.HomeMode := mcHOME_DIRECT;
				axis.ctrl.BasicControl.Parameter.HomePosition := 0;
				axis.ctrl.Cmd := CONST.AXIS.CALIBR;(* Achse referenzieren*)
				state := ST_CALIBR_WAIT;
			ELSIF powerbridge.pressurepresent THEN
				err.text := 'Stanze steht unter Druck';
				err.state := state;
				state := ST_ERROR;
			ELSIF axis.ctrl.MC_ReadStatus_0.Errorstop THEN //die Achse geht in ErrorStop wenn die sichere Geschwindigkeit überschritten wird
				//			err.text := 'Werkzeug falsch parametriert';
				//			err.fnc := 'MC_Home';
				//			err.set := TRUE;
				//			err.state := state;
				err := axis.ctrl.err;
				state := ST_ERROR;
			ELSIF cmd = CONST.CUTTINGUNIT.CMDs.NO_CMD THEN
				state := ST_QUIT;
			END_IF

		ST_CALIBR_WAIT://22
			axis.refSwitchConfig();
			IF axis.ctrl.BasicControl.AxisState.Homed AND(data.recipe.mode = CONST.CUTTINGUNIT.MODEs.SYNC_RUN OR data.recipe.mode = CONST.CUTTINGUNIT.MODEs.CROSS_CUT) THEN
				axis.refSwitchConfig(Enable := FALSE);
				cmd := CONST.CUTTINGUNIT.CMDs.NO_CMD;
				status.isCalibrated := TRUE;(* Achse ist referenziert*)
				state := ST_CALIBR_START_NULLPOS;
			ELSIF axis.ctrl.BasicControl.AxisState.Homed AND data.recipe.mode = CONST.CUTTINGUNIT.MODEs.FREE_RUN THEN
				axis.refSwitchConfig(Enable := FALSE);
				cmd := CONST.CUTTINGUNIT.CMDs.NO_CMD;
				status.isCalibrated := TRUE;
				state := ST_CALIBR_WAIT_NULLPOS;//da keine Bewegung notwendig
			ELSIF axis.ctrl.MC_ReadStatus_0.Disabled AND cmd = CONST.CUTTINGUNIT.CMDs.SETDATA THEN
				state := ST_SETDATA_WAIT;
			ELSIF axis.ctrl.MC_ReadStatus_0.Errorstop THEN //die Achse geht in ErrorStop wenn die sichere Geschwindigkeit überschritten wird
				err.text := 'Werkzeug falsch parametriert';
				err.fnc := 'MC_Home';
				err.set := TRUE;
				err.state := state;
				state := ST_ERROR;
			ELSIF cmd <> CONST.CUTTINGUNIT.CMDs.CALIBR THEN //Stanze beim Referenzieren stoppen
				axis.ctrl.Cmd := CONST.AXIS.STOP;
				IF NOT axis.ctrl.busy THEN
					axis.ctrl.Cmd := CONST.AXIS.NOACTION;
					state := ST_QUIT;	(*abwarten bis die Achse nicht busy ist*)
				END_IF
			END_IF

		ST_CALIBR_START_NULLPOS://24
			IF cmd = CONST.CUTTINGUNIT.CMDs.ABORT THEN
				state := ST_ABORT;
			ELSIF axis.ctrl.busy OR axis.ctrl.Cmd <> CONST.AXIS.NOACTION THEN
				axis.ctrl(Cmd := CONST.AXIS.NOACTION);
			ELSIF  NOT axis.ctrl.busy THEN(* jetzt halbe Drehung vorfahren*)
				axis.ctrl.Position := 1000; // 1mm da der Sensor oben sitzt
				axis.ctrl.Acceleration := 120000;
				axis.ctrl.Deceleration := 120000;
				axis.ctrl.Velocity :=1.7;
				axis.ctrl.Cmd := CONST.AXIS.SETPOS;
				state := ST_CALIBR_WAIT_NULLPOS;
				(* Homeposition ist wo das Werkzeug/Blech den Anfang hat da darf korregiert werden*)
			END_IF

		ST_CALIBR_WAIT_NULLPOS://26
			IF NOT axis.ctrl.busy THEN
				IF status.isCalibrated THEN // 13.03.15 Stanze ist referenziert dann koppeln
					axis.ctrl.Cmd := CONST.AXIS.NOACTION;
					cmd := CONST.CUTTINGUNIT.CMDs.CPL_ON;
					state := ST_GENERATE_TABLE_START;
				ELSIF NOT status.isCalibrated THEN
					axis.ctrl.Cmd := CONST.AXIS.NOACTION;
					state := ST_QUIT;
				END_IF
			ELSIF axis.ctrl.MC_ReadStatus_0.Errorstop THEN //Achse hat einen Fehler
				err := axis.ctrl.err;
				err.state := state;
				state := ST_ERROR;
			END_IF

		ST_GENERATE_TABLE_START: //35
			IF  cmd = CONST.CUTTINGUNIT.CMDs.CPL_ON OR cmdtmp = CONST.CUTTINGUNIT.CMDs.CPL_ON THEN //cmdtmp fürs automatisches Koppeln
				IF axis.ctrl.MC_ReadStatus_0.StandStill OR axis.ctrl.MC_ReadStatus_0.Disabled THEN
					camtable.index := 3;
					axis.cplCam.Execute := FALSE;
					camtable.createCam := TRUE;
					state := ST_GENERATE_TABLE_WAIT;
				ELSIF axis.ctrl.MC_ReadStatus_0.SynchronizedMotion THEN //19.02.15
					state := ST_QUIT;
				ELSIF axis.ctrl.MC_ReadStatus_0.Error OR axis.ctrl.MC_ReadStatus_0.Errorstop THEN
					err.set := TRUE;
					err.state := ST_GENERATE_TABLE_START;
					err.fnc := 'FB_CuttingConfig';
					state := ST_ERROR;
				END_IF
			ELSE
				state := ST_QUIT;
			END_IF

		ST_GENERATE_TABLE_WAIT://36
			camtable(AxisREF := axis.ctrl.AxisREF, CONST := CONST, MasterAxisREF := machineMaster.AxisREF, data := data, scalePerimeter:= scalePerimeter,  Name := status.name );
			IF camtable.done THEN
				camtable.createCam := FALSE;
				state := ST_CPL_TABLE_START;
			ELSIF camtable.err.flag THEN
				err := camtable.err;
				err();
				state := ST_ERROR;
			END_IF

		ST_CPL_TABLE_START: //37
			camtable((*createCam := FALSE,*)CONST := CONST, AxisREF := axis.ctrl.AxisREF, MasterAxisREF := machineMaster.AxisREF, data := data, scalePerimeter:= scalePerimeter,  Name := status.name );
			IF axis.ctrl.MC_ReadStatus_0.StandStill  AND camtable.camTableID > 0 AND NOT camtable.done THEN
				axis.cplCam.Master :=  machineMaster.AxisREF;
				axis.cplCam.Slave := axis.ctrl.AxisREF;
				axis.cplCam.StartMode :=  mcDIRECT;
				axis.cplCam.MasterOffset := 0;// machineMaster.MC_ReadActualPosition_0.Position;(*pMasterAxis.monitor.s mach keinen Sinn da die Kurvenscheibe periodisch ist*) ;
				axis.cplCam.SlaveOffset := 0;
				axis.cplCam.MasterScaling := 1;
				axis.cplCam.SlaveScaling  := 1;
				axis.cplCam.CamTableID  := camtable.camTableID (*1*);
				state := ST_CPL_EXECUTE;
			ELSIF NOT axis.ctrl.MC_ReadStatus_0.StandStill THEN
				state := ST_QUIT;
			ELSIF axis.cplCam.Error THEN
				err(set := TRUE ,fnc := 'FB_CuttinConfig' ,text := 'MC_CamIn', state := ST_CPL_TABLE_START, id :=  axis.cplCam.ErrorID);
				axis.cplCam.Execute := FALSE;
				state := ST_ERROR;
			ELSIF camtable.camTableID = 0 THEN
				err(set := TRUE ,fnc := 'FB_CuttinConfig' ,text := 'camtable', state := ST_CPL_TABLE_START, id :=  camtable.err.id);
				state := ST_ERROR;
			END_IF

		ST_CPL_CAMTABLE://38
			axis.cplCam( Master :=  machineMaster.AxisREF, Slave := axis.ctrl.AxisREF);
			axis.cplCam.Execute := TRUE;
			IF axis.ctrl.MC_ReadStatus_0.SynchronizedMotion THEN
				axis.cplCam.Execute := FALSE;
				cmd := CONST.CUTTINGUNIT.CMDs.NO_CMD;
				state := ST_QUIT;
			ELSIF axis.cplCam.Error THEN
				axis.cplCam.Execute := FALSE;
				err(set := TRUE ,fnc := 'FB_CuttinConfig' ,text := 'MC_CamIn', state := ST_CPL_TABLE_START, id :=  axis.cplCam.ErrorID);
				state := ST_ERROR;
			ELSIF axis.cplCam.CommandAborted THEN
				axis.cplCam.Execute := FALSE;
				state := ST_CPL_EXECUTE;
			END_IF

		ST_CPL_EXECUTE: //39
			axis.cplCam( Master :=  machineMaster.AxisREF, Slave := axis.ctrl.AxisREF);
			axis.cplCam.Execute := FALSE;
			state := ST_CPL_CAMTABLE;

		ST_CPLOFF_START://80 (* bei B&R funktioniert der MC_gearout nur mit MC_Gearin deshalb MC_stop*)
			IF cmd = CONST.CUTTINGUNIT.CMDs.ABORT THEN
				state := ST_ABORT;
			ELSIF axis.ctrl.MC_ReadStatus_0.SynchronizedMotion  THEN
				axis.MC_BR_Phasing_0 (Enable := FALSE, InitData := FALSE);
				IF NOT 	axis.MC_BR_Phasing_0.Busy THEN
					axis.ctrl.Cmd := CONST.AXIS.STOP;
					IF axis.ctrl.busy THEN
						state := ST_CPLOFF_WAIT;
					END_IF
				END_IF
			ELSIF axis.ctrl.MC_ReadStatus_0.StandStill THEN
				IF NOT axis.ctrl.busy THEN
					state := ST_CPLOFF_WAIT;
				END_IF
			END_IF

		ST_CPLOFF_WAIT://81
			IF  axis.ctrl.MC_ReadStatus_0.StandStill AND cmd = CONST.CUTTINGUNIT.CMDs.NO_CMD THEN
				axis.ctrl.Cmd := CONST.AXIS.NOACTION;
				status.isCoupled := FALSE;
				status.isSynchronized := FALSE;
			ELSIF cmdtmp = CONST.CUTTINGUNIT.CMDs.SETDATA THEN
				axis.ctrl.Cmd := CONST.AXIS.NOACTION;
				status.isCalibrated := FALSE;
				status.isCoupled := FALSE;
				status.isSynchronized := FALSE;
				state := ST_SETDATA_START;
			ELSIF cmdtmp = CONST.CUTTINGUNIT.CMDs.CALIBR THEN
				axis.ctrl.Cmd := CONST.AXIS.NOACTION;
				status.isCalibrated := FALSE;
				status.isCoupled := FALSE;
				status.isSynchronized := FALSE;
				state := ST_SETDATA_START;
			ELSIF cmdtmp = CONST.CUTTINGUNIT.CMDs.INIT THEN
				status.isCalibrated := FALSE;
				status.isCoupled := FALSE;
				status.isSynchronized := FALSE;
				axis.ctrl.Cmd := CONST.AXIS.NOACTION;
				state := ST_INIT_START;
			ELSIF cmdtmp = CONST.CUTTINGUNIT.CMDs.DEINIT THEN
				axis.ctrl.Cmd := CONST.AXIS.NOACTION;
				status.isCalibrated := FALSE;
				status.isCoupled := FALSE;
				status.isSynchronized := FALSE;
				state := ST_DEINIT_CPLSLAVEOFF_START;
			ELSIF cmdtmp = CONST.CUTTINGUNIT.CMDs.SYNC THEN
				status.isCoupled := FALSE;
				status.isSynchronized := FALSE;
				state := ST_SYNC_START;
			ELSIF axis.ctrl.MC_ReadStatus_0.StandStill AND NOT axis.ctrl.busy AND cmd = CONST.CUTTINGUNIT.CMDs.MOVEBW THEN
				axis.ctrl.Cmd := CONST.AXIS.NOACTION;
				state := ST_MOVE_START;
			ELSIF axis.ctrl.MC_ReadStatus_0.StandStill AND NOT axis.ctrl.busy  AND cmd = CONST.CUTTINGUNIT.CMDs.MOVEFW THEN
				axis.ctrl.Cmd := CONST.AXIS.NOACTION;
				state := ST_MOVE_START;
			ELSE
				state := ST_QUIT;
			END_IF

		ST_DEINIT_CPLSLAVEOFF_START://67
			IF status.isCoupled THEN
				state := ST_CPLOFF_START;
			ELSE
				state := ST_DEINIT;
			END_IF

		ST_DEINIT:
			IF NOT axis.ctrl.busy THEN
				IF axis.ctrl.MC_ReadStatus_0.Error OR axis.ctrl.MC_ReadStatus_0.Errorstop  THEN
					err.state := state;
					state := ST_ERROR;
				ELSE
					status.isInitialized := FALSE;
					status.isSynchronized := FALSE;
					status.isCalibrated := FALSE;
					IF cmdtmp = CONST.CUTTINGUNIT.CMDs.SETDATA THEN
						state := ST_SETDATA_START;
					ELSIF cmdtmp = CONST.CUTTINGUNIT.CMDs.CALIBR THEN
						state := ST_SETDATA_START;
					ELSIF cmdtmp = CONST.CUTTINGUNIT.CMDs.INIT THEN
						axis.ctrl.Cmd := CONST.AXIS.NOACTION;
						state := ST_INIT_START;
					ELSE
						axis.ctrl.Cmd := CONST.AXIS.POWER_OFF;
						IF NOT axis.ctrl.busy THEN
							axis.ctrl.Cmd := CONST.AXIS.NOACTION;
							state := ST_QUIT;
						END_IF
					END_IF
				END_IF
			END_IF

//		ST_MOVE_START:// 40 falls die Achse nicht initialisiert ist
//			IF axis.ctrl.MC_ReadStatus_0.SynchronizedMotion THEN
//				state:= ST_CPLOFF_START;
//			ELSIF NOT axis.MC_BR_Phasing_0.Busy  AND axis.ctrl.MC_ReadStatus_0.StandStill AND cmd <>  CONST.CUTTINGUNIT.CMDs.NO_CMD  THEN
//				IF cmd = CONST.CUTTINGUNIT.CMDs.MOVEBW THEN
//					axis.ctrl(Cmd := CONST.AXIS.JOG_NEG, Velocity := 3, Acceleration := 120000, Deceleration := 120000,);
//				ELSIF cmd = CONST.CUTTINGUNIT.CMDs.MOVEFW THEN
//					axis.ctrl(Cmd := CONST.AXIS.JOG_POS, Velocity := 3, Acceleration := 120000, Deceleration := 120000);
//				END_IF
//			ELSIF cmd =  CONST.CUTTINGUNIT.CMDs.NO_CMD THEN
//				axis.ctrl(Cmd := CONST.AXIS.NOACTION );
//				state := ST_MOVE_QUIT;
//			END_IF

//***********************neu********************// OKrebs 14.01.16
		ST_MOVE_START:// 40 falls die Achse nicht initialisiert ist
			IF powerbridge.pressurepresent THEN
			err.set := TRUE;
			err.text := 'cutteraxis unter Druck';
			err.state := state;
			(*	powerbridge.bridgedownbutton.buttonDown.LDT.button := TRUE; *)
			//				state := ST_ERROR;
			ELSIF NOT axis.MC_BR_Phasing_0.Busy  AND axis.ctrl.MC_ReadStatus_0.SynchronizedMotion AND cmd <>  CONST.CUTTINGUNIT.CMDs.NO_CMD AND NOT powerbridge.pressurepresent THEN
				IF cmd = CONST.CUTTINGUNIT.CMDs.MOVEBW THEN
					axis.MC_BR_Phasing_0.Acceleration := 90000;
					axis.MC_BR_Phasing_0.ApplicationMode := mcVELOCITY_CONTROL ;
					axis.MC_BR_Phasing_0.Slave := axis.ctrl.AxisREF;
					axis.MC_BR_Phasing_0.Velocity := - 16666.67 * 3; //1m/min
					axis.MC_BR_Phasing_0.Enable := TRUE;
					axis.MC_BR_Phasing_0.InitData := TRUE;
					axis.MC_BR_Phasing_0.PerformVelocityControl := TRUE;
				ELSIF cmd = CONST.CUTTINGUNIT.CMDs.MOVEFW (*AND TON_0.Q*) THEN
					axis.MC_BR_Phasing_0.Acceleration := 90000;
					axis.MC_BR_Phasing_0.ApplicationMode := mcVELOCITY_CONTROL;
					axis.MC_BR_Phasing_0.Slave := axis.ctrl.AxisREF;
					axis.MC_BR_Phasing_0.Velocity := 16666.67 * 3; //1m/min
					axis.MC_BR_Phasing_0.Enable := TRUE;
					axis.MC_BR_Phasing_0.InitData := TRUE;
					axis.MC_BR_Phasing_0.PerformVelocityControl := TRUE;
				END_IF
			ELSIF NOT axis.MC_BR_Phasing_0.Busy  AND axis.ctrl.MC_ReadStatus_0.StandStill AND cmd <>  CONST.CUTTINGUNIT.CMDs.NO_CMD AND NOT powerbridge.pressurepresent THEN
				IF cmd = CONST.CUTTINGUNIT.CMDs.MOVEBW THEN
					axis.ctrl(Cmd := CONST.AXIS.JOG_NEG, Velocity := 3, Acceleration := 120000, Deceleration := 120000);
				ELSIF cmd = CONST.CUTTINGUNIT.CMDs.MOVEFW THEN
					axis.ctrl(Cmd := CONST.AXIS.JOG_POS, Velocity := 3, Acceleration := 120000, Deceleration := 120000);
				END_IF
			ELSIF cmd =  CONST.CUTTINGUNIT.CMDs.NO_CMD AND axis.ctrl.MC_ReadStatus_0.SynchronizedMotion THEN
				axis.MC_BR_Phasing_0.Velocity := 0;
				axis.MC_BR_Phasing_0.PerformVelocityControl := FALSE;
				axis.MC_BR_Phasing_0.InitData := FALSE;
				IF axis.MC_BR_Phasing_0.ShiftAttained THEN
					axis.MC_BR_Phasing_0.Enable := FALSE;
					state := ST_QUIT;
				END_IF
			ELSIF cmd =  CONST.CUTTINGUNIT.CMDs.NO_CMD AND (axis.ctrl.MC_ReadStatus_0.StandStill OR axis.ctrl.MC_ReadStatus_0.ContinuousMotion) THEN
				axis.ctrl(Cmd := CONST.AXIS.NOACTION);
				state := ST_QUIT;
			ELSIF  axis.ctrl.MC_ReadStatus_0.Disabled THEN
				state := ST_QUIT;
			ELSE

			END_IF

//******************************************************************************

		ST_MOVE_WAIT:
			axis.ctrl();
			IF cmd = CONST.CUTTINGUNIT.CMDs.NO_CMD THEN
				axis.ctrl(Cmd := CONST.AXIS.NOACTION );
				state := ST_MOVE_QUIT;
			END_IF
		//
		ST_MOVE_QUIT: (* hier evtl. koppeln*)
			//		IF axis.ctrl.MC_ReadStatus_0.StandStill OR axis.ctrl.MC_ReadStatus_0.Errorstop
			//			OR axis.ctrl.MC_ReadStatus_0.StandStill OR axis.ctrl.MC_ReadStatus_0.Error THEN
			//			state := ST_QUIT;
			IF data.recipe.mode = CONST.CUTTINGUNIT.MODEs.DISABLE THEN //AW 19.05.15
				state := ST_QUIT;//Wenn Stanze nicht aktiv dann nicht koppeln
			ELSIF data.recipe.mode = CONST.CUTTINGUNIT.MODEs.FREE_RUN OR data.recipe.mode = CONST.CUTTINGUNIT.MODEs.SYNC_RUN OR
				data.recipe.mode = CONST.CUTTINGUNIT.MODEs.CROSS_CUT THEN
				cmd := CONST.CUTTINGUNIT.CMDs.CPL_ON;
				cmdtmp := cmd;
				state := ST_GENERATE_TABLE_START;
			END_IF

		ST_CPL_WAIT:
			axis.cplCam( Master :=  machineMaster.AxisREF, Slave := axis.ctrl.AxisREF);
			IF axis.cplCam.Busy AND axis.ctrl.MC_ReadStatus_0.SynchronizedMotion THEN
				axis.cplCam( Execute := FALSE, Master :=  machineMaster.AxisREF, Slave := axis.ctrl.AxisREF);
				status.isCoupled := TRUE;
				state := ST_QUIT;
			ELSIF axis.cplCam.Error THEN
				err.id := axis.cplCam.ErrorID;
				err.fnc := 'axis.cplCam';
				err.state := state;
				state := ST_ERROR;
			END_IF
		//
		ST_SYNC_START://70
			timer(PT := T#2s);
			axis.MC_BR_Phasing_0.Enable := FALSE;
			axis.MC_BR_Phasing_0.InitData := FALSE;
			getNextUnitSyncPos(machineMaster := machineMaster, uAxis := axis.ctrl, markpoints := markpoints,
			uData := data, scalePerimeter := scalePerimeter, setCutOffset := setCutOffset, CONST := CONST);
			syncDiff := getNextUnitSyncPos.syncDataBefore.correctionNoLimit;
			IF cmd = CONST.CUTTINGUNIT.CMDs.ABORT THEN
				state := ST_ABORT;
			ELSIF NOT machineMaster.MC_ReadStatus_0.StandStill THEN
				err.set := TRUE;
				err.state := state;
				err.text := 'MasterModulAxis steht nicht';
				state := ST_ERROR;
			ELSIF powerbridge.pressurepresent AND NOT timer.Q THEN
				err.set := TRUE;
				err.text := 'cutteraxis unter Druck';
				err.state := state;
			(*	powerbridge.bridgedownbutton.buttonDown.LDT.button := TRUE; *)
				timer.IN := TRUE;
//				state := ST_ERROR;
			ELSIF timer.IN AND timer.Q THEN
				timer.IN := FALSE;
			ELSIF axis.ctrl.MC_ReadStatus_0.SynchronizedMotion AND NOT powerbridge.pressurepresent AND NOT axis.MC_BR_Phasing_0.Active AND NOT axis.MC_BR_Phasing_0.Busy AND syncDiff <> 0 AND NOT timer.Q THEN
				//				getNextUnitSyncPos(machineMaster := machineMaster, uAxis := axis.ctrl, markpoints := markpoints,
				//									uData := data, scalePerimeter := scalePerimeter, setCutOffset := setCutOffset);
				//				syncDiff := getNextUnitSyncPos.syncDataBefore.correctionNoLimit;
				//				IF syncDiff < -0.1 OR syncDiff > 0.1 THEN
				getNextUnitSyncPos.trigger := TRUE;
				axis.MC_BR_Phasing_0.Enable := TRUE;
				axis.MC_BR_Phasing_0.Acceleration := 90000;
				axis.MC_BR_Phasing_0.ApplicationDistance := scalePerimeter.realperimeter;
				axis.MC_BR_Phasing_0.ApplicationMode := mcTIME_BASED;//1;//mcMASTER_POSITION_BASED;
				axis.MC_BR_Phasing_0.Slave := axis.ctrl.AxisREF;
				axis.MC_BR_Phasing_0.ShiftMode := mcRELATIVE;//1
				axis.MC_BR_Phasing_0.Velocity := 16666.67; //1m/min
				axis.MC_BR_Phasing_0.Shift := syncDiff;// zu korregierende Strecke
				axis.MC_BR_Phasing_0.InitData := TRUE;
				err.text := '';
				state := ST_SYNC_START_CORRECTION;

			ELSIF syncDiff = 0 (*AND NOT axis.ctrl.MC_ReadStatus_0.SynchronizedMotion *)THEN //beim ersten Durchlauf wenn keine Marken eingelesen war
				err(set := TRUE, fnc := 'FB_CuttingConfig',text := 'Kein Synchroner Punkt-Marken, neue einlesen', state := ST_SYNC_START);
				state := ST_QUIT;
			ELSIF  axis.ctrl.MC_ReadStatus_0.StandStill THEN //Stanze nicht ist gekoppelt keine Aufsynchronisation möglich
				state := ST_QUIT;
			END_IF

		ST_SYNC_START_CORRECTION: //73

			IF  axis.MC_BR_Phasing_0.Active THEN
				state := ST_SYNC_WAIT_CORRECTION;
			ELSIF axis.MC_BR_Phasing_0.Error THEN
				err(set := TRUE, fnc := 'MC_BR_Phasing_0 in FB_CuttingConfig',text := 'MC_BR_Phasing_0', state := ST_SYNC_START_CORRECTION, id := axis.MC_BR_Phasing_0.ErrorID);
				axis.MC_BR_Phasing_0.InitData := FALSE;
				state := ST_ERROR;
			END_IF
		//
		ST_SYNC_WAIT_CORRECTION://74
			IF axis.MC_BR_Phasing_0.ShiftAttained THEN
				axis.MC_BR_Phasing_0.InitData := FALSE;
				axis.MC_BR_Phasing_0.Enable := FALSE;
				status.isSynchronized := TRUE;
				getNextUnitSyncPos(machineMaster := machineMaster,
								uAxis := axis.ctrl,
								markpoints := markpoints,
								uData := data,
								scalePerimeter := scalePerimeter,
								setCutOffset := setCutOffset, CONST := CONST);
				cmd := CONST.CUTTINGUNIT.CMDs.NO_CMD;

				state := ST_QUIT;
			ELSIF axis.MC_BR_Phasing_0.Error THEN
				err(set := TRUE, fnc := 'MC_BR_Phasing_0 in FB_CuttingConfig',text := 'MC_BR_Phasing_0', state := ST_SYNC_START_CORRECTION, id := axis.MC_BR_Phasing_0.ErrorID);
				axis.MC_BR_Phasing_0.InitData := FALSE;
				state := ST_ERROR;
			END_IF

		ST_ERROR:
			err();
			IF LEN(err.fnc) < 1 THEN
				err.fnc := 'FB_CuttingConfig';
			END_IF
			IF cmd = CONST.CUTTINGUNIT.CMDs.RESET THEN
				axis.cplCam( Execute := FALSE, Master :=  machineMaster.AxisREF, Slave := axis.ctrl.AxisREF);
				axis.MC_BR_Phasing_0.Enable := FALSE;
				axis.MC_BR_Phasing_0.InitData:= FALSE;
				InitAxisSubjectPar(Axis := axis.ctrl.AxisREF, Subject := ncDIG_IN,Execute := FALSE);
				axis.ctrl(Cmd := CONST.AXIS.RESET);
				err(reset:= TRUE);
				state := ST_ABORT_QUIT;
			END_IF

		ST_ABORT:
			state := ST_ABORT_QUIT;

		ST_ABORT_QUIT:
			IF NOT axis.ctrl.busy THEN
				axis.ctrl(Cmd := CONST.AXIS.NOACTION);
				cmd := CONST.CUTTINGUNIT.CMDs.NO_CMD;
				state := ST_QUIT;
			END_IF

		ST_QUIT:
			IF cmd = CONST.CUTTINGUNIT.CMDs.ABORT THEN
				busy := TRUE;
				state := ST_ABORT;
			ELSE
				busy := FALSE;
				IF cmd <> CONST.CUTTINGUNIT.CMDs.NO_CMD THEN
					axis.ctrl.Cmd := CONST.AXIS.NOACTION;
					state := ST_IDLE;
				END_IF

			END_IF

	END_CASE
	axis.MC_BR_Phasing_0();
	InitAxisSubjectPar.Axis := axis.ctrl.AxisREF;
	InitAxisSubjectPar();

END_FUNCTION_BLOCK
```

#### FB_CutterAxis.st
```iecst
(********************************************************************
 * COPYRIGHT -- Microsoft
 ********************************************************************
 * Programm: MAIN
 * Datei: FB_CutterAxis.st
 * Autor: Awalz
 * Erstellt: 19. Mai 2014
 ********************************************************************
 * Implementierung des Programms MAIN
 ********************************************************************)

 (*<$Description$> TODO: Bitte Kommentar hier einzufügen </$Description$>*)
FUNCTION_BLOCK FB_CutterAxis
END_FUNCTION_BLOCK
```

#### FB_CuttingUnit.st
```iecst
(********************************************************************
 * COPYRIGHT -- Microsoft
 ********************************************************************
 * Programm: MAIN
 * Datei: FB_CuttingUnit.st
 * Autor: Awalz
 * Erstellt: 19. Mai 2014
 ********************************************************************
 * Implementierung des Programms MAIN
 ********************************************************************)

 (*<$Description$> TODO: Bitte Kommentar hier einzufügen </$Description$>*)
FUNCTION_BLOCK FB_CuttingUnit
END_FUNCTION_BLOCK
```

#### FB_CuttingCheckData.st
```iecst
(********************************************************************
 * COPYRIGHT -- Microsoft
 ********************************************************************
 * Programm: MAIN
 * Datei: FB_CuttingUnitCheckData.st
 * Autor: okrebs
 * Erstellt: 23. Mai 2014
 ********************************************************************
 * Implementierung des Programms MAIN
 ********************************************************************)

(* TODO: Bitte Kommentar hier einzufügen *)
FUNCTION_BLOCK FB_CuttingCheckData
//
	err(reset := TRUE);
	tmpString := '';
	IF modeCtrl.mode = CONST.CUTTINGUNIT.MODEs.DISABLE THEN
		;
	ELSIF modeCtrl.mode = CONST.CUTTINGUNIT.MODEs.FREE_RUN OR modeCtrl.mode = CONST.CUTTINGUNIT.MODEs.SYNC_RUN THEN
		IF (*recipe.toolNumber < CONST.CUTTINGUNIT.TOOLs.MIN_TOOLS OR*) recipe.toolNumber > CONST.CUTTINGUNIT.TOOLs.MAX_TOOLS THEN
			err.flag := TRUE;
			tmpString := USINT_TO_STRING(recipe.toolNumber);
		(*	tmpString := CONCAT( 'ToolNr: ', tmpString );*)
			err.text := 'Fehler: Produktdaten.';
			err.id := CONST.CUTTINGUNIT.ERRORs.RECIPE_TOOLNR;
		ELSE

			IF  (recipe.tool.cutEndPosition < recipe.tool.cutStartPosition) OR (recipe.tool.cutEndPosition > general.periodLength)
					OR (recipe.tool.cutStartPosition > general.periodLength) THEN
				err.flag := TRUE;
				err.text := 'Fehler: Produktdaten. Kontur Beschreibung';
				err.id := CONST.CUTTINGUNIT.ERRORs.RECIPE_SHAPE_CONFIG;
				err.fnc := 'FB_CuttingUnitChkData';
			END_IF
			IF recipe.tool.cogCutting < 3 THEN
				err.flag := TRUE;
				tmpString := INT_TO_STRING(recipe.toolNumber);
				err.text := 'Fehler: Zähneanzahl CutterWerkzeug:';
				err.id := CONST.CUTTINGUNIT.ERRORs.CUTTER_ZAEHNE;
				err.fnc := 'FB_CuttingUnitChkData';
			END_IF
			IF recipe.tool.cogSupportSpindle < 3 THEN
				err.flag := TRUE;
				tmpString := INT_TO_STRING(recipe.toolNumber);
				err.text :='Fehler: Zähneanzahl GegenwalzeWerkzeug:';
				err.id := CONST.CUTTINGUNIT.ERRORs.ANVILROLLER_ZAEHNE;
				err.fnc := 'FB_CuttingUnitChkData';
			END_IF
		END_IF
	ELSE
		err.flag := TRUE;
		err.text := 'Fehler: Produktdaten Betriebsart undefiniert';
		err.id := CONST.CUTTINGUNIT.ERRORs.RECIPE_MODE_UNDEF;
		err.fnc := 'FB_CuttingUnitChkData';
	END_IF

END_FUNCTION_BLOCK
```

#### FB_CUTTINGUNIT_DATA.st
```iecst
(********************************************************************
 * COPYRIGHT -- Microsoft
 ********************************************************************
 * Programm: MAIN
 * Datei: FB_CUTTINGUNIT_DATA.st
 * Autor: Awalz
 * Erstellt: 3. Juni 2014
 ********************************************************************
 * Implementierung des Programms MAIN
 ********************************************************************)

 (*<$Description$> TODO: Bitte Kommentar hier einzufügen </$Description$>*)
FUNCTION_BLOCK FB_CUTTINGUNIT_DATA

//	tmpData(compare := TRUE,BetrCtrl := BetrCtrl );
//	IF tmpData.changed THEN
//		set := TRUE;
//	ELSIF tmpData.err.flag THEN
//			set := FALSE;
//	ELSIF tmpData.changed AND NOT tmpData.err.flag THEN
//		newRecipe:= TRUE;
//		newMach:=TRUE;
//		newTools:= TRUE;
//		machdata :=	tmpData.setMach;
//		recipe := tmpData.setRecipe;
//		general := tmpData.setMasterModulData;
//	ELSE
//		newRecipe:= FALSE;
//		newMach:=FALSE;
//		newTools:= FALSE;
//	END_IF
END_FUNCTION_BLOCK
```

#### FB_CUTTINGUNIT_TMPDATA.st
```iecst
(********************************************************************
 * COPYRIGHT -- Microsoft
 ********************************************************************
 * Programm: MAIN
 * Datei: FB_CUTTINGUNIT_TMPDATA.st
 * Autor: Awalz
 * Erstellt: 3. Juni 2014
 ********************************************************************
 * Implementierung des Programms MAIN
 ********************************************************************)

 (*<$Description$> TODO: Bitte Kommentar hier einzufügen </$Description$>*)
FUNCTION_BLOCK FB_CUTTINGUNIT_TMPDATA
	IF BetrCtrl.value = CONST.MACHINEMODES.MANUAL THEN
		IF set THEN
			actMasterModulData := setMasterModulData;
			actMach := setMach;
			actRecipe := setRecipe;
			set := FALSE;
		END_IF
	ELSE
		err.flag := TRUE;
		err.text := 'Rezept nicht geladen Maschine ist in Aotomatikmodus';
		err.fnc := 'FB_CUTTINGUNIT_TMPDATA';
		err.set := TRUE;
	END_IF

	changed := FALSE;
	changedText := '';
	IF compare THEN
		IF actMasterModulData.periodLength <> setMasterModulData.periodLength THEN
			changed := TRUE;
			changedText := 'MasterModulData.recipe.periodLength';
		ELSIF actRecipe.mode <> setRecipe.mode THEN
			changed := TRUE;
			changedText := 'Recipe.mode';
		ELSIF actRecipe.toolNumber <> setRecipe.toolNumber THEN
			changed := TRUE;
			changedText := 'Recipe.toolNumber';
		ELSIF actRecipe.tool.cogSupportSpindle <> setRecipe.tool.cogSupportSpindle  THEN
			changed := TRUE;
			changedText := 'Tool.anvilroller.zaehne';
		ELSIF actRecipe.tool.description <> setRecipe.tool.description THEN
			changed := TRUE;
			changedText := 'Tool.arrangementSpecial';
		ELSIF actRecipe.tool.gearRatioMotor <> setRecipe.tool.gearRatioMotor THEN
			changed := TRUE;
			changedText := 'Tool.gearFactorModule';
		ELSIF actRecipe.tool.cutStartPosition <> setRecipe.tool.cutStartPosition THEN
			changed := TRUE;
			changedText := 'Tool.cutStartPosition';
		ELSIF actRecipe.tool.numberToolSegments <> setRecipe.tool.numberToolSegments  THEN
			changed := TRUE;
			changedText := 'Tool.numberToolsegments';
		ELSIF actRecipe.tool.cogCutting <> setRecipe.tool.cogCutting THEN
			changed := TRUE;
			changedText := 'Tool.cutter.zaehne';
		ELSIF actRecipe.tool.cutEndPosition <> setRecipe.tool.cutEndPosition THEN
			changed := TRUE;
			changedText := 'Tool.cutEndPosition';
		ELSE
//			syncPosCmp(actSyncPos := actTool.shape.syncPos, setSyncPos := setTool.shape.syncPos);
//			IF syncPosCmp.changed THEN
//				changed := TRUE;
//				changedText := CONCAT('Tool.shape.', syncPosCmp.changedText);
//			END_IF
		END_IF
	END_IF
END_FUNCTION_BLOCK
```

#### Package Logical/MainMachineCtrl/MAIN/CuttingUnit/Functions - Paket

#### FB_GetCuttingMark.st
```iecst
(********************************************************************
 * COPYRIGHT -- Nitto
 ********************************************************************
 * Programm: MAIN
 * Datei: FB_GetCuttingMark.st
 * Autor: s_spilker
 * Erstellt: 9. November 2015
 ********************************************************************
 * Implementierung des Programms MAIN
 ********************************************************************)

(* TODO: Bitte Kommentar hier einfügen *)
FUNCTION_BLOCK FB_GetCuttingMark
	unitPos := uData.machdata.position - usercorrec - uData.recipe.RmOffset -248000;//214000;
	myRefposition := uData.machdata.position + markpoints.RegMarkPosition; // da der Wert negativ ist
	pMasterAxisREF ACCESS machineMaster.AxisREF;
	masterPos := pMasterAxisREF.monitor.s;
	pSlaveAxisREF ACCESS uAxis.AxisREF;
	markBefore();
	markAfter();
	IF unitPos < myRefposition THEN (* Cuttingunit vor dem Markpoint Sensor *)
		configError := TRUE;
	ELSE
		configError := FALSE;
	END_IF
	IF markpoints.markpointlist.valid THEN
		(* Position Masters bzw des Druckmarke stellt die flißende bewegung der Druckmarke zu aufgenommenen Stelle*)
		actMarkDiff:= pMasterAxisREF.monitor.s - markpoints.MC_BR_TouchProbe_0.RecordedValue;
		(* myRefpogen ist die Position des Druckmarkensensors bez zu Einheitosition*)
		absMarkPos := myRefposition + actMarkDiff;(*ab den Nulldurchgang der Stanze wird der Wert positiv*)
		IF absMarkPos < unitPos THEN
//			IF ABS (markpoints.RegMarkPosition)> uData.general.periodLength THEN
//				diffToUnitBefore := absMarkPos - unitPos;// diffToUnitBefore muss immer negativ sein
//			ELSE
				diffToUnitBefore := absMarkPos - unitPos;// - uData.general.periodLength;
		(*	END_IF*)
		ELSE
			diffToUnitAfter := absMarkPos - unitPos;
		END_IF
	END_IF
END_FUNCTION_BLOCK
```

#### FB_SyncData.st
```iecst
(********************************************************************
 * COPYRIGHT -- Nitto
 ********************************************************************
 * Programm: MAIN
 * Datei: FB_SyncData.st
 * Autor: s_spilker
 * Erstellt: 9. November 2015
 ********************************************************************
 * Implementierung des Programms MAIN
 ********************************************************************)

(* TODO: Bitte Kommentar hier einfügen *)
FUNCTION_BLOCK FB_SyncData
END_FUNCTION_BLOCK
```

#### FB_CuttingCamCtrl.st
```iecst
(********************************************************************
 * COPYRIGHT -- Microsoft
 ********************************************************************
 * Programm: MAIN
 * Datei: FB_CuttingCamCtrl.st
 * Autor: awalz
 * Erstellt: 20. Juli 2014
 ********************************************************************
 * Implementierung des Programms MAIN
 ********************************************************************)

(* TODO: Bitte Kommentar hier einfügen *)
FUNCTION_BLOCK FB_CuttingCamCtrl
	getNextUnitSyncPos (uData := data, machineMaster := machineMaster,  markpoints := markpoints, uAxis := axis.ctrl, scalePerimeter := scalePerimeter, setCutOffset := setCutOffset, CONST := CONST);
	syncData := getNextUnitSyncPos.syncDataBefore;

	CASE state OF
		0:
			IF enable THEN
				IF axis.ctrl.MC_ReadStatus_0.SynchronizedMotion THEN
					axis.MC_BR_Phasing_0(Enable := FALSE,Slave:=axis.ctrl.AxisREF);
					IF syncData.markIndx <> actSyncPosIdent THEN
						axis.MC_BR_Phasing_0.Enable 		:= TRUE;
						axis.MC_BR_Phasing_0.Velocity		:= LIMIT (30000, (machineMaster.MC_ReadActualVelocity_0.Velocity ), 1000000);
						axis.MC_BR_Phasing_0.Acceleration 	:= 2500000; (*150000;*)
						IF ABS (syncData.correctionNoLimit) < 1000 THEN // wenn die Abweichung kleiner als 1mm dann synchronisiert melden
							status.isSynchronized := TRUE;
						ELSE
							status.isSynchronized := FALSE;
						END_IF
						////					(*DAs Phasing geschieht in scalePerimeter.ToolSegmentPeriod - 120000 | -120000 um dem System zeit zu gebne das Erfolgreiche Phasen zu erfassen und für ein erneutes bereit zu sein *)
						axis.MC_BR_Phasing_0.ApplicationDistance :=  data.general.periodLength -30000;//   scalePerimeter.ToolSegmentPeriod - 20000;
						axis.MC_BR_Phasing_0.ApplicationMode	:= mcMASTER_DISTANCE_BASED (*mcMASTER_POSITION_BASED*);
						axis.MC_BR_Phasing_0.ShiftMode		:= mcRELATIVE(*mcABSOLUTE*);
						axis.MC_BR_Phasing_0.Shift 			:= LIMIT (-data.recipe.MaxCorr, syncData.correctionNoLimit,data.recipe.MaxCorr);
						axis.MC_BR_Phasing_0.InitData 		:= TRUE;
						(*	IF axis.MC_BR_Offset_0.DataInitialized THEN*)
						actSyncPosIdent := syncData.markIndx;
						usercorrtemp	:= 	usercorrection;
						counter := counter + 1;
						state := 1;
						(*END_IF*)
					END_IF
				END_IF

			END_IF

		1:	IF enable THEN
				IF 	axis.MC_BR_Phasing_0.ShiftAttained THEN
					donecounter := donecounter + 1;
					axis.MC_BR_Phasing_0.InitData := FALSE;
					axis.MC_BR_Phasing_0.Enable := FALSE;
					shiftValuetmp := axis.MC_BR_Phasing_0.ActualShiftValue;
					state := 0;
				ELSIF axis.MC_BR_Phasing_0.Error THEN
					axis.MC_BR_Phasing_0.InitData := FALSE;
					axis.MC_BR_Phasing_0.Enable 	:= FALSE;
					errorcounter := errorcounter + 1;
					state := 0;
				END_IF
			ELSE
				axis.MC_BR_Phasing_0.InitData := FALSE;
				axis.MC_BR_Phasing_0.Enable := FALSE;
				shiftValuetmp := axis.MC_BR_Phasing_0.ActualShiftValue;
				errorcounter := errorcounter + 1;
				state := 0;
			END_IF

	END_CASE
	axis.MC_BR_Phasing_0();
END_FUNCTION_BLOCK
```

#### FB_WriteEncoder.st
```iecst
(********************************************************************
 * COPYRIGHT -- Microsoft
 ********************************************************************
 * Programm: MAIN
 * Datei: FB_WriteEncoder.st
 * Autor: Awalz
 * Erstellt: 23. Mai 2014
 ********************************************************************
 * Implementierung des Programms MAIN
 ********************************************************************)

 (*<$Description$> TODO: Bitte Kommentar hier einzufügen </$Description$>*)
FUNCTION_BLOCK FB_WriteEncoder
	MC_ReadStatus_0.Axis	:= AxisREF;
	MC_ReadStatus_0.Enable	:= NOT MC_ReadStatus_0.Error;
	MC_ReadStatus_0();

	MC_BR_ReadDriveStatus_0.Axis			:= AxisREF;
	MC_BR_ReadDriveStatus_0.AdrDriveStatus	:= ADR(DriveStatus);
	MC_BR_ReadDriveStatus_0.Enable			:= NOT MC_BR_ReadDriveStatus_0.Error;
	MC_BR_ReadDriveStatus_0();

	MC_BR_InitModPos_0.Axis				:= AxisREF;
	MC_BR_InitModPos_0();
	pAxis ACCESS AxisREF;
	EncIf_Act.scaling.load.rev_motor 	:= pAxis.encoder_if.parameter.scaling.load.rev_motor;
	EncIf_Act.scaling.load.units 		:= pAxis.encoder_if.parameter.scaling.load.units;
	CASE state OF

		ST_IDLE: IF enable THEN
				IF check THEN
					busy := TRUE;
//					scalePerimeter.realperimeter := UINT_TO_REAL (data.recipe.tool.cogCutting )* data.recipe.tool.cogmodul * 1000;
//					scalePerimeter.NumberToolSegments := MAX (1, data.recipe.tool.numberToolSegments);
					scalePerimeter();
//					EncIf_Set.scaling.load.rev_motor 	:= data.recipe.tool.gearRatioMotor * data.recipe.tool.cogCutting;
//					EncIf_Set.scaling.load.units 		:= data.recipe.tool.cogSupportSpindle * scalePerimeter.Scaledperimeter;
					EncIf_InitValid := TRUE;
					state :=  ST_SET_MODULO;

				END_IF

			END_IF

		ST_SETDATA_START://1

		ST_SETDATA_WAIT://2

		ST_SET_MODULO://3

			ModPeriod_Set	:= scalePerimeter.ToolSegmentPeriod;
			IF  ModPeriod_Set = MC_BR_InitModPos_0.Period THEN
				state := ST_QUIT; (* wenn gleiche Periode dann Periode icht ändern*)
			END_IF
			IF 0 < ModPeriod_Set < brmldexp( 2, 23) AND DriveStatus.NetworkInit AND(MC_ReadStatus_0.Disabled OR MC_ReadStatus_0.StandStill) AND  EncIf_InitValid THEN
				(*warum zwanzig RS FBs wo ist der Sinn*)
				MC_BR_InitModPos_0.Factor	:= 1;
				MC_BR_InitModPos_0.Execute	:= TRUE;
				MC_BR_InitModPos_0.Period	:= ModPeriod_Set;
				(*	MC_BR_InitModPos_0();*)
				EncIf_InitValid := FALSE;
			END_IF;
			//complete modulo period setup by copying the downloaded parameters into the "Act" structure
			IF MC_BR_InitModPos_0.Done THEN
				ModPeriod_Act	:= MC_BR_InitModPos_0.Period;
				MC_BR_InitModPos_0.Execute	:= FALSE;
				EncIf_InitValid := TRUE;
				state := ST_QUIT;
			ELSIF MC_BR_InitModPos_0.Error THEN
				err.fnc := 'FB_WriteEncoder';
				err.text := 'Modulo Achse';
				err.state := ST_SETDATA_WAIT;
				err.id := MC_BR_InitModPos_0.ErrorID;
				err.set := TRUE;
				state := ST_ERROR;
			END_IF;

		ST_ERROR: //5
			IF LEN(err.fnc) < 1 THEN
				err.fnc := 'FB_WriteEncoder';
				err.text := ' Werkzeugdaten sind falsch';
			END_IF
			err(set := TRUE);
			state := ST_QUIT;

		ST_QUIT://6
			check := FALSE;
			busy := FALSE;
			state := ST_IDLE;
	END_CASE

END_FUNCTION_BLOCK
```

#### FB_CuttingModeCtrl.st
```iecst
(********************************************************************
 * COPYRIGHT -- Microsoft
 ********************************************************************
 * Programm: MAIN
 * Datei: FB_Cuttingmode.st
 * Autor: Awalz
 * Erstellt: 20. Mai 2014
 ********************************************************************
 * Implementierung des Programms MAIN
 ********************************************************************)

 (*<$Description$> TODO: Bitte Kommentar hier einzufügen </$Description$>*)
FUNCTION_BLOCK FB_CuttingModeCtrl

	CASE state OF
		ST_IDLE_BEFORE:
			busy := FALSE;
			state := ST_IDLE;

		ST_IDLE:
			IF mode <> CONST.CUTTINGUNIT.MODEs.DISABLE THEN
				busy := TRUE;
				err(reset := TRUE);
				IF axis.ctrl.MC_ReadStatus_0.SynchronizedMotion THEN
					IF mode = CONST.CUTTINGUNIT.MODEs.FREE_RUN THEN
						state := ST_FREECUTTING_BEFORE;
					ELSIF mode = CONST.CUTTINGUNIT.MODEs.SYNC_RUN THEN
						state := ST_SYNCCUTTING_BEFORE;
					END_IF
				END_IF
		END_IF

		ST_IDLE_QUIT:
			busy := FALSE;
			IF mode = CONST.CUTTINGUNIT.MODEs.DISABLE THEN
				err(reset := TRUE);
				state := ST_IDLE_BEFORE;
			END_IF

		ST_FREECUTTING_BEFORE:
			busy := FALSE;
			state := ST_FREECUTTING;

		ST_FREECUTTING:
			IF mode <> CONST.CUTTINGUNIT.MODEs.FREE_RUN THEN
				camCtrl(enable := FALSE, machineMaster := machineMaster, axis := axis, scalePerimeter := scalePerimeter, data := data, status := status,
						markpoints := markpoints, getNextUnitSyncPos := getNextUnitSyncPos, setCutOffset := setCutOffset, CONST := CONST);
				busy := TRUE;
				err(reset := TRUE);
				IF mode = CONST.CUTTINGUNIT.MODEs.DISABLE THEN
					state := ST_IDLE_BEFORE;
				ELSIF mode = CONST.CUTTINGUNIT.MODEs.SYNC_RUN THEN
					state := ST_SYNCCUTTING_BEFORE;
				END_IF
			ELSE
				camCtrl(enable := TRUE, machineMaster := machineMaster, axis := axis, scalePerimeter := scalePerimeter, data := data, status := status,
						markpoints := markpoints, getNextUnitSyncPos := getNextUnitSyncPos, setCutOffset := setCutOffset, CONST := CONST);
			END_IF;

		ST_SYNCCUTTING_BEFORE:
	//		status.mode.set(value := CONST.CUTTINGUNIT.MODEs.SYNC_RUN);
	//		SetGearRatio(GearRatio := 1, Slave := masterAxis.ctrl.ref );
			busy := FALSE;
			state := ST_SYNCCUTTING;

		ST_SYNCCUTTING:
			IF mode <> CONST.CUTTINGUNIT.MODEs.SYNC_RUN THEN
				busy := TRUE;
				state := ST_SYNCCUTTING_AFTER;
			ELSE
				camCtrl(enable := TRUE, machineMaster := machineMaster, axis := axis, scalePerimeter := scalePerimeter, data := data, status := status,
						markpoints := markpoints, getNextUnitSyncPos := getNextUnitSyncPos, setCutOffset := setCutOffset, CONST := CONST);

			END_IF

		ST_SYNCCUTTING_AFTER:
			camCtrl(enable := FALSE, machineMaster := machineMaster, axis := axis, scalePerimeter := scalePerimeter, data := data, status := status,
						markpoints := markpoints, getNextUnitSyncPos := getNextUnitSyncPos, setCutOffset := setCutOffset, CONST := CONST);
			state := ST_IDLE;

	END_CASE
END_FUNCTION_BLOCK
```
